  LIN {X 4999.921,Y 0.097,Z -215.600,A 90.00334,B 0.00000,C 180.00000} ; insert
  LIN {X 4999.921,Y 0.097,Z -215.600,A 90.00334,B 0.00000,C 180.00000} ; release
  LIN {X 4999.921,Y 0.097,Z 84.400,A 90.00334,B 0.00000,C 180.00000} ; retreat
  ; Step 681, bar 945
  LIN {X 5015.921,Y 0.097,Z 947.280,A 90.00334,B 0.00000,C 180.00000} ; outside
  LIN {X 5015.921,Y 0.097,Z 34.400,A 90.00334,B 0.00000,C 180.00000} ; preinsert
  LIN {X 5015.921,Y 0.097,Z -215.600,A 90.00334,B 0.00000,C 180.00000} ; insert
  LIN {X 5015.921,Y 0.097,Z -215.600,A 90.00334,B 0.00000,C 180.00000} ; release
  LIN {X 5015.921,Y 0.097,Z 84.400,A 90.00334,B 0.00000,C 180.00000} ; retreat
  ; Step 682, bar 943
  LIN {X 5124.921,Y 0.097,Z 947.280,A 90.00334,B 0.00000,C 180.00000} ; outside
  LIN {X 5124.921,Y 0.097,Z 34.400,A 90.00334,B 0.00000,C 180.00000} ; preinsert
  LIN {X 5124.921,Y 0.097,Z -215.600,A 90.00334,B 0.00000,C 180.00000} ; insert
  LIN {X 5124.921,Y 0.097,Z -215.600,A 90.00334,B 0.00000,C 180.00000} ; release
  LIN {X 5124.921,Y 0.097,Z 84.400,A 90.00334,B 0.00000,C 180.00000} ; retreat
  ; Step 683, bar 946
  LIN {X 5249.921,Y 0.097,Z 947.280,A 90.00334,B 0.00000,C 180.00000} ; outside
  LIN {X 5249.921,Y 0.097,Z 34.400,A 90.00334,B 0.00000,C 180.00000} ; preinsert
  LIN {X 5249.921,Y 0.097,Z -215.600,A 90.00334,B 0.00000,C 180.00000} ; insert
  LIN {X 5249.921,Y 0.097,Z -215.600,A 90.00334,B 0.00000,C 180.00000} ; release
  LIN {X 5249.921,Y 0.097,Z 84.400,A 90.00334,B 0.00000,C 180.00000} ; retreat
  ; Step 684, bar 947
  LIN {X 5374.921,Y 0.097,Z 947.280,A 90.00334,B 0.00000,C 180.00000} ; outside
  LIN {X 5374.921,Y 0.097,Z 34.400,A 90.00334,B 0.00000,C 180.00000} ; preinsert
  LIN {X 5374.921,Y 0.097,Z -215.600,A 90.00334,B 0.00000,C 180.00000} ; insert
  LIN {X 5374.921,Y 0.097,Z -215.600,A 90.00334,B 0.00000,C 180.00000} ; release
  LIN {X 5374.921,Y 0.097,Z 84.400,A 90.00334,B 0.00000,C 180.00000} ; retreat
  ; Step 685, bar 949
  LIN {X 5499.921,Y 0.097,Z 947.280,A 90.00334,B 0.00000,C 180.00000} ; outside
  LIN {X 5499.921,Y 0.097,Z 34.400,A 90.00334,B 0.00000,C 180.00000} ; preinsert
  LIN {X 5499.921,Y 0.097,Z -215.600,A 90.00334,B 0.00000,C 180.00000} ; insert
  LIN {X 5499.921,Y 0.097,Z -215.600,A 90.00334,B 0.00000,C 180.00000} ; release
  LIN {X 5499.921,Y 0.097,Z 84.400,A 90.00334,B 0.00000,C 180.00000} ; retreat
  ; Step 686, bar 950
  LIN {X 5515.921,Y 0.097,Z 947.280,A 90.00334,B 0.00000,C 180.00000} ; outside
  LIN {X 5515.921,Y 0.097,Z 34.400,A 90.00334,B 0.00000,C 180.00000} ; preinsert
  LIN {X 5515.921,Y 0.097,Z -215.600,A 90.00334,B 0.00000,C 180.00000} ; insert
  LIN {X 5515.921,Y 0.097,Z -215.600,A 90.00334,B 0.00000,C 180.00000} ; release
  LIN {X 5515.921,Y 0.097,Z 84.400,A 90.00334,B 0.00000,C 180.00000} ; retreat
  ; Step 687, bar 948
  LIN {X 5624.921,Y 0.097,Z 947.280,A 90.00334,B 0.00000,C 180.00000} ; outside
  LIN {X 5624.921,Y 0.097,Z 34.400,A 90.00334,B 0.00000,C 180.00000} ; preinsert
  LIN {X 5624.921,Y 0.097,Z -215.600,A 90.00334,B 0.00000,C 180.00000} ; insert
  LIN {X 5624.921,Y 0.097,Z -215.600,A 90.00334,B 0.00000,C 180.00000} ; release
  LIN {X 5624.921,Y 0.097,Z 84.400,A 90.00334,B 0.00000,C 180.00000} ; retreat
  ; Step 688, bar 951
  LIN {X 5749.921,Y 0.097,Z 947.280,A 90.00334,B 0.00000,C 180.00000} ; outside
  LIN {X 5749.921,Y 0.097,Z 34.400,A 90.00334,B 0.00000,C 180.00000} ; preinsert
  LIN {X 5749.921,Y 0.097,Z -215.600,A 90.00334,B 0.00000,C 180.00000} ; insert
  LIN {X 5749.921,Y 0.097,Z -215.600,A 90.00334,B 0.00000,C 180.00000} ; release
  LIN {X 5749.921,Y 0.097,Z 84.400,A 90.00334,B 0.00000,C 180.00000} ; retreat
  ; Step 689, bar 954
  LIN {X 5874.921,Y 0.097,Z 947.280,A 90.00334,B 0.00000,C 180.00000} ; outside
  LIN {X 5874.921,Y 0.097,Z 34.400,A 90.00334,B 0.00000,C 180.00000} ; preinsert
  LIN {X 5874.921,Y 0.097,Z -215.600,A 90.00334,B 0.00000,C 180.00000} ; insert
  LIN {X 5874.921,Y 0.097,Z -215.600,A 90.00334,B 0.00000,C 180.00000} ; release
  LIN {X 5874.921,Y 0.097,Z 84.400,A 90.00334,B 0.00000,C 180.00000} ; retreat
  ; Step 690, bar 955
  LIN {X 5890.921,Y 0.097,Z 947.280,A 90.00334,B 0.00000,C 180.00000} ; outside
  LIN {X 5890.921,Y 0.097,Z 34.400,A 90.00334,B 0.00000,C 180.00000} ; preinsert
  LIN {X 5890.921,Y 0.097,Z -215.600,A 90.00334,B 0.00000,C 180.00000} ; insert
  LIN {X 5890.921,Y 0.097,Z -215.600,A 90.00334,B 0.00000,C 180.00000} ; release
  LIN {X 5890.921,Y 0.097,Z 84.400,A 90.00334,B 0.00000,C 180.00000} ; retreat
  ; Step 691, bar 952
  LIN {X 5999.921,Y 0.097,Z 947.280,A 90.00334,B 0.00000,C 180.00000} ; outside
  LIN {X 5999.921,Y 0.097,Z 34.400,A 90.00334,B 0.00000,C 180.00000} ; preinsert
  LIN {X 5999.921,Y 0.097,Z -215.600,A 90.00334,B 0.00000,C 180.00000} ; insert
  LIN {X 5999.921,Y 0.097,Z -215.600,A 90.00334,B 0.00000,C 180.00000} ; release
  LIN {X 5999.921,Y 0.097,Z 84.400,A 90.00334,B 0.00000,C 180.00000} ; retreat
  ; Step 692, bar 953
  LIN {X 6124.921,Y 0.097,Z 947.280,A 90.00334,B 0.00000,C 180.00000} ; outside
  LIN {X 6124.921,Y 0.097,Z 34.400,A 90.00334,B 0.00000,C 180.00000} ; preinsert
  LIN {X 6124.921,Y 0.097,Z -215.600,A 90.00334,B 0.00000,C 180.00000} ; insert
  LIN {X 6124.921,Y 0.097,Z -215.600,A 90.00334,B 0.00000,C 180.00000} ; release
  LIN {X 6124.921,Y 0.097,Z 84.400,A 90.00334,B 0.00000,C 180.00000} ; retreat
  ; Step 693, bar 956
  LIN {X 6249.921,Y 0.097,Z 947.280,A 90.00334,B 0.00000,C 180.00000} ; outside
  LIN {X 6249.921,Y 0.097,Z 34.400,A 90.00334,B 0.00000,C 180.00000} ; preinsert
  LIN {X 6249.921,Y 0.097,Z -215.600,A 90.00334,B 0.00000,C 180.00000} ; insert
  LIN {X 6249.921,Y 0.097,Z -215.600,A 90.00334,B 0.00000,C 180.00000} ; release
  LIN {X 6249.921,Y 0.097,Z 84.400,A 90.00334,B 0.00000,C 180.00000} ; retreat
  ; Step 694, bar 957
  LIN {X 6374.921,Y 0.097,Z 947.280,A 90.00334,B 0.00000,C 180.00000} ; outside
  LIN {X 6374.921,Y 0.097,Z 34.400,A 90.00334,B 0.00000,C 180.00000} ; preinsert
  LIN {X 6374.921,Y 0.097,Z -215.600,A 90.00334,B 0.00000,C 180.00000} ; insert
  LIN {X 6374.921,Y 0.097,Z -215.600,A 90.00334,B 0.00000,C 180.00000} ; release
  LIN {X 6374.921,Y 0.097,Z 84.400,A 90.00334,B 0.00000,C 180.00000} ; retreat
  ; Step 695, bar 959
  LIN {X 6499.921,Y 0.097,Z 947.280,A 90.00334,B 0.00000,C 180.00000} ; outside
  LIN {X 6499.921,Y 0.097,Z 34.400,A 90.00334,B 0.00000,C 180.00000} ; preinsert
  LIN {X 6499.921,Y 0.097,Z -215.600,A 90.00334,B 0.00000,C 180.00000} ; insert
  LIN {X 6499.921,Y 0.097,Z -215.600,A 90.00334,B 0.00000,C 180.00000} ; release
  LIN {X 6499.921,Y 0.097,Z 84.400,A 90.00334,B 0.00000,C 180.00000} ; retreat
  ; Step 696, bar 960
  LIN {X 6515.921,Y 0.097,Z 947.280,A 90.00334,B 0.00000,C 180.00000} ; outside
  LIN {X 6515.921,Y 0.097,Z 34.400,A 90.00334,B 0.00000,C 180.00000} ; preinsert
  LIN {X 6515.921,Y 0.097,Z -215.600,A 90.00334,B 0.00000,C 180.00000} ; insert
  LIN {X 6515.921,Y 0.097,Z -215.600,A 90.00334,B 0.00000,C 180.00000} ; release
  LIN {X 6515.921,Y 0.097,Z 84.400,A 90.00334,B 0.00000,C 180.00000} ; retreat
  ; Step 697, bar 958
  LIN {X 6624.921,Y 0.097,Z 947.280,A 90.00334,B 0.00000,C 180.00000} ; outside
  LIN {X 6624.921,Y 0.097,Z 34.400,A 90.00334,B 0.00000,C 180.00000} ; preinsert
  LIN {X 6624.921,Y 0.097,Z -215.600,A 90.00334,B 0.00000,C 180.00000} ; insert
  LIN {X 6624.921,Y 0.097,Z -215.600,A 90.00334,B 0.00000,C 180.00000} ; release
  LIN {X 6624.921,Y 0.097,Z 84.400,A 90.00334,B 0.00000,C 180.00000} ; retreat
  ; Step 698, bar 961
  LIN {X 6749.921,Y 0.097,Z 947.280,A 90.00334,B 0.00000,C 180.00000} ; outside
  LIN {X 6749.921,Y 0.097,Z 34.400,A 90.00334,B 0.00000,C 180.00000} ; preinsert
  LIN {X 6749.921,Y 0.097,Z -215.600,A 90.00334,B 0.00000,C 180.00000} ; insert
  LIN {X 6749.921,Y 0.097,Z -215.600,A 90.00334,B 0.00000,C 180.00000} ; release
  LIN {X 6749.921,Y 0.097,Z 84.400,A 90.00334,B 0.00000,C 180.00000} ; retreat
  ; Step 699, bar 962
  LIN {X 6874.921,Y 0.097,Z 947.280,A 90.00334,B 0.00000,C 180.00000} ; outside
  LIN {X 6874.921,Y 0.097,Z 34.400,A 90.00334,B 0.00000,C 180.00000} ; preinsert
  LIN {X 6874.921,Y 0.097,Z -215.600,A 90.00334,B 0.00000,C 180.00000} ; insert
  LIN {X 6874.921,Y 0.097,Z -215.600,A 90.00334,B 0.00000,C 180.00000} ; release
  LIN {X 6874.921,Y 0.097,Z 84.400,A 90.00334,B 0.00000,C 180.00000} ; retreat
  ; Step 700, bar 964
  LIN {X 6999.921,Y 0.097,Z 947.280,A 90.00334,B 0.00000,C 180.00000} ; outside
  LIN {X 6999.921,Y 0.097,Z 34.400,A 90.00334,B 0.00000,C 180.00000} ; preinsert
  LIN {X 6999.921,Y 0.097,Z -215.600,A 90.00334,B 0.00000,C 180.00000} ; insert
  LIN {X 6999.921,Y 0.097,Z -215.600,A 90.00334,B 0.00000,C 180.00000} ; release
  LIN {X 6999.921,Y 0.097,Z 84.400,A 90.00334,B 0.00000,C 180.00000} ; retreat
  ; Step 701, bar 965
  LIN {X 7015.921,Y 0.097,Z 947.280,A 90.00334,B 0.00000,C 180.00000} ; outside
  LIN {X 7015.921,Y 0.097,Z 34.400,A 90.00334,B 0.00000,C 180.00000} ; preinsert
  LIN {X 7015.921,Y 0.097,Z -215.600,A 90.00334,B 0.00000,C 180.00000} ; insert
  LIN {X 7015.921,Y 0.097,Z -215.600,A 90.00334,B 0.00000,C 180.00000} ; release
  LIN {X 7015.921,Y 0.097,Z 84.400,A 90.00334,B 0.00000,C 180.00000} ; retreat
  ; Step 702, bar 963
  LIN {X 7124.921,Y 0.097,Z 947.280,A 90.00334,B 0.00000,C 180.00000} ; outside
  LIN {X 7124.921,Y 0.097,Z 34.400,A 90.00334,B 0.00000,C 180.00000} ; preinsert
  LIN {X 7124.921,Y 0.097,Z -215.600,A 90.00334,B 0.00000,C 180.00000} ; insert
  LIN {X 7124.921,Y 0.097,Z -215.600,A 90.00334,B 0.00000,C 180.00000} ; release
  LIN {X 7124.921,Y 0.097,Z 84.400,A 90.00334,B 0.00000,C 180.00000} ; retreat
  ; Step 703, bar 966
  LIN {X 7249.921,Y 0.097,Z 947.280,A 90.00334,B 0.00000,C 180.00000} ; outside
  LIN {X 7249.921,Y 0.097,Z 34.400,A 90.00334,B 0.00000,C 180.00000} ; preinsert
  LIN {X 7249.921,Y 0.097,Z -215.600,A 90.00334,B 0.00000,C 180.00000} ; insert
  LIN {X 7249.921,Y 0.097,Z -215.600,A 90.00334,B 0.00000,C 180.00000} ; release
  LIN {X 7249.921,Y 0.097,Z 84.400,A 90.00334,B 0.00000,C 180.00000} ; retreat
  ; Step 704, bar 967
  LIN {X 7374.921,Y 0.097,Z 947.280,A 90.00334,B 0.00000,C 180.00000} ; outside
  LIN {X 7374.921,Y 0.097,Z 34.400,A 90.00334,B 0.00000,C 180.00000} ; preinsert
  LIN {X 7374.921,Y 0.097,Z -215.600,A 90.00334,B 0.00000,C 180.00000} ; insert
  LIN {X 7374.921,Y 0.097,Z -215.600,A 90.00334,B 0.00000,C 180.00000} ; release
  LIN {X 7374.921,Y 0.097,Z 84.400,A 90.00334,B 0.00000,C 180.00000} ; retreat
  ; Step 705, bar 969
  LIN {X 7499.921,Y 0.097,Z 947.280,A 90.00334,B 0.00000,C 180.00000} ; outside
  LIN {X 7499.921,Y 0.097,Z 34.400,A 90.00334,B 0.00000,C 180.00000} ; preinsert
  LIN {X 7499.921,Y 0.097,Z -215.600,A 90.00334,B 0.00000,C 180.00000} ; insert
  LIN {X 7499.921,Y 0.097,Z -215.600,A 90.00334,B 0.00000,C 180.00000} ; release
  LIN {X 7499.921,Y 0.097,Z 84.400,A 90.00334,B 0.00000,C 180.00000} ; retreat
  ; Step 706, bar 970
  LIN {X 7515.921,Y 0.097,Z 947.280,A 90.00334,B 0.00000,C 180.00000} ; outside
  LIN {X 7515.921,Y 0.097,Z 34.400,A 90.00334,B 0.00000,C 180.00000} ; preinsert
  LIN {X 7515.921,Y 0.097,Z -215.600,A 90.00334,B 0.00000,C 180.00000} ; insert
  LIN {X 7515.921,Y 0.097,Z -215.600,A 90.00334,B 0.00000,C 180.00000} ; release
  LIN {X 7515.921,Y 0.097,Z 84.400,A 90.00334,B 0.00000,C 180.00000} ; retreat
  ; Step 707, bar 968
  LIN {X 7624.921,Y 0.097,Z 947.280,A 90.00334,B 0.00000,C 180.00000} ; outside
  LIN {X 7624.921,Y 0.097,Z 34.400,A 90.00334,B 0.00000,C 180.00000} ; preinsert
  LIN {X 7624.921,Y 0.097,Z -215.600,A 90.00334,B 0.00000,C 180.00000} ; insert
  LIN {X 7624.921,Y 0.097,Z -215.600,A 90.00334,B 0.00000,C 180.00000} ; release
  LIN {X 7624.921,Y 0.097,Z 84.400,A 90.00334,B 0.00000,C 180.00000} ; retreat
  ; Step 708, bar 971
  LIN {X 7749.921,Y 0.097,Z 947.280,A 90.00334,B 0.00000,C 180.00000} ; outside
  LIN {X 7749.921,Y 0.097,Z 34.400,A 90.00334,B 0.00000,C 180.00000} ; preinsert
  LIN {X 7749.921,Y 0.097,Z -215.600,A 90.00334,B 0.00000,C 180.00000} ; insert
  LIN {X 7749.921,Y 0.097,Z -215.600,A 90.00334,B 0.00000,C 180.00000} ; release
  LIN {X 7749.921,Y 0.097,Z 84.400,A 90.00334,B 0.00000,C 180.00000} ; retreat
  ; Step 709, bar 972
  LIN {X 7874.921,Y 0.097,Z 947.280,A 90.00334,B 0.00000,C 180.00000} ; outside
  LIN {X 7874.921,Y 0.097,Z 34.400,A 90.00334,B 0.00000,C 180.00000} ; preinsert
  LIN {X 7874.921,Y 0.097,Z -215.600,A 90.00334,B 0.00000,C 180.00000} ; insert
  LIN {X 7874.921,Y 0.097,Z -215.600,A 90.00334,B 0.00000,C 180.00000} ; release
  LIN {X 7874.921,Y 0.097,Z 84.400,A 90.00334,B 0.00000,C 180.00000} ; retreat
  ; Step 710, bar 974
  LIN {X 7999.921,Y 0.097,Z 947.280,A 90.00334,B 0.00000,C 180.00000} ; outside
  LIN {X 7999.921,Y 0.097,Z 34.400,A 90.00334,B 0.00000,C 180.00000} ; preinsert
  LIN {X 7999.921,Y 0.097,Z -215.600,A 90.00334,B 0.00000,C 180.00000} ; insert
  LIN {X 7999.921,Y 0.097,Z -215.600,A 90.00334,B 0.00000,C 180.00000} ; release
  LIN {X 7999.921,Y 0.097,Z 84.400,A 90.00334,B 0.00000,C 180.00000} ; retreat
  ; Step 711, bar 975
  LIN {X 8015.921,Y 0.097,Z 947.280,A 90.00334,B 0.00000,C 180.00000} ; outside
  LIN {X 8015.921,Y 0.097,Z 34.400,A 90.00334,B 0.00000,C 180.00000} ; preinsert
  LIN {X 8015.921,Y 0.097,Z -215.600,A 90.00334,B 0.00000,C 180.00000} ; insert
  LIN {X 8015.921,Y 0.097,Z -215.600,A 90.00334,B 0.00000,C 180.00000} ; release
  LIN {X 8015.921,Y 0.097,Z 84.400,A 90.00334,B 0.00000,C 180.00000} ; retreat
  ; Step 712, bar 973
  LIN {X 8124.921,Y 0.097,Z 947.280,A 90.00334,B 0.00000,C 180.00000} ; outside
  LIN {X 8124.921,Y 0.097,Z 34.400,A 90.00334,B 0.00000,C 180.00000} ; preinsert
  LIN {X 8124.921,Y 0.097,Z -215.600,A 90.00334,B 0.00000,C 180.00000} ; insert
  LIN {X 8124.921,Y 0.097,Z -215.600,A 90.00334,B 0.00000,C 180.00000} ; release
  LIN {X 8124.921,Y 0.097,Z 84.400,A 90.00334,B 0.00000,C 180.00000} ; retreat
  ; Step 713, bar 976
  LIN {X 8249.921,Y 0.097,Z 947.280,A 90.00334,B 0.00000,C 180.00000} ; outside
  LIN {X 8249.921,Y 0.097,Z 34.400,A 90.00334,B 0.00000,C 180.00000} ; preinsert
  LIN {X 8249.921,Y 0.097,Z -215.600,A 90.00334,B 0.00000,C 180.00000} ; insert
  LIN {X 8249.921,Y 0.097,Z -215.600,A 90.00334,B 0.00000,C 180.00000} ; release
  LIN {X 8249.921,Y 0.097,Z 84.400,A 90.00334,B 0.00000,C 180.00000} ; retreat
  ; Step 714, bar 977
  LIN {X 8374.921,Y 0.097,Z 947.280,A 90.00334,B 0.00000,C 180.00000} ; outside
  LIN {X 8374.921,Y 0.097,Z 34.400,A 90.00334,B 0.00000,C 180.00000} ; preinsert
  LIN {X 8374.921,Y 0.097,Z -215.600,A 90.00334,B 0.00000,C 180.00000} ; insert
  LIN {X 8374.921,Y 0.097,Z -215.600,A 90.00334,B 0.00000,C 180.00000} ; release
  LIN {X 8374.921,Y 0.097,Z 84.400,A 90.00334,B 0.00000,C 180.00000} ; retreat
  ; Step 715, bar 979
  LIN {X 8499.921,Y 0.097,Z 947.280,A 90.00334,B 0.00000,C 180.00000} ; outside
  LIN {X 8499.921,Y 0.097,Z 34.400,A 90.00334,B 0.00000,C 180.00000} ; preinsert
  LIN {X 8499.921,Y 0.097,Z -215.600,A 90.00334,B 0.00000,C 180.00000} ; insert
  LIN {X 8499.921,Y 0.097,Z -215.600,A 90.00334,B 0.00000,C 180.00000} ; release
  LIN {X 8499.921,Y 0.097,Z 84.400,A 90.00334,B 0.00000,C 180.00000} ; retreat
  ; Step 716, bar 980
  LIN {X 8515.921,Y 0.097,Z 947.280,A 90.00334,B 0.00000,C 180.00000} ; outside
  LIN {X 8515.921,Y 0.097,Z 34.400,A 90.00334,B 0.00000,C 180.00000} ; preinsert
  LIN {X 8515.921,Y 0.097,Z -215.600,A 90.00334,B 0.00000,C 180.00000} ; insert
  LIN {X 8515.921,Y 0.097,Z -215.600,A 90.00334,B 0.00000,C 180.00000} ; release
  LIN {X 8515.921,Y 0.097,Z 84.400,A 90.00334,B 0.00000,C 180.00000} ; retreat
  ; Step 717, bar 978
  LIN {X 8624.921,Y 0.097,Z 947.280,A 90.00334,B 0.00000,C 180.00000} ; outside
  LIN {X 8624.921,Y 0.097,Z 34.400,A 90.00334,B 0.00000,C 180.00000} ; preinsert
  LIN {X 8624.921,Y 0.097,Z -215.600,A 90.00334,B 0.00000,C 180.00000} ; insert
  LIN {X 8624.921,Y 0.097,Z -215.600,A 90.00334,B 0.00000,C 180.00000} ; release
  LIN {X 8624.921,Y 0.097,Z 84.400,A 90.00334,B 0.00000,C 180.00000} ; retreat
  ; Step 718, bar 981
  LIN {X 8749.921,Y 0.097,Z 947.280,A 90.00334,B 0.00000,C 180.00000} ; outside
  LIN {X 8749.921,Y 0.097,Z 34.400,A 90.00334,B 0.00000,C 180.00000} ; preinsert
  LIN {X 8749.921,Y 0.097,Z -215.600,A 90.00334,B 0.00000,C 180.00000} ; insert
  LIN {X 8749.921,Y 0.097,Z -215.600,A 90.00334,B 0.00000,C 180.00000} ; release
  LIN {X 8749.921,Y 0.097,Z 84.400,A 90.00334,B 0.00000,C 180.00000} ; retreat
  ; Step 719, bar 982
  LIN {X 8874.921,Y 0.097,Z 947.280,A 90.00334,B 0.00000,C 180.00000} ; outside
  LIN {X 8874.921,Y 0.097,Z 34.400,A 90.00334,B 0.00000,C 180.00000} ; preinsert
  LIN {X 8874.921,Y 0.097,Z -215.600,A 90.00334,B 0.00000,C 180.00000} ; insert
  LIN {X 8874.921,Y 0.097,Z -215.600,A 90.00334,B 0.00000,C 180.00000} ; release
  LIN {X 8874.921,Y 0.097,Z 84.400,A 90.00334,B 0.00000,C 180.00000} ; retreat
  ; Step 720, bar 984
  LIN {X 8999.921,Y 0.097,Z 947.280,A 90.00334,B 0.00000,C 180.00000} ; outside
  LIN {X 8999.921,Y 0.097,Z 34.400,A 90.00334,B 0.00000,C 180.00000} ; preinsert
  LIN {X 8999.921,Y 0.097,Z -215.600,A 90.00334,B 0.00000,C 180.00000} ; insert
  LIN {X 8999.921,Y 0.097,Z -215.600,A 90.00334,B 0.00000,C 180.00000} ; release
  LIN {X 8999.921,Y 0.097,Z 84.400,A 90.00334,B 0.00000,C 180.00000} ; retreat
  ; Step 721, bar 985
  LIN {X 9015.921,Y 0.097,Z 947.280,A 90.00334,B 0.00000,C 180.00000} ; outside
  LIN {X 9015.921,Y 0.097,Z 34.400,A 90.00334,B 0.00000,C 180.00000} ; preinsert
  LIN {X 9015.921,Y 0.097,Z -215.600,A 90.00334,B 0.00000,C 180.00000} ; insert
  LIN {X 9015.921,Y 0.097,Z -215.600,A 90.00334,B 0.00000,C 180.00000} ; release
  LIN {X 9015.921,Y 0.097,Z 84.400,A 90.00334,B 0.00000,C 180.00000} ; retreat
  ; Step 722, bar 983
  LIN {X 9124.921,Y 0.097,Z 947.280,A 90.00334,B 0.00000,C 180.00000} ; outside
  LIN {X 9124.921,Y 0.097,Z 34.400,A 90.00334,B 0.00000,C 180.00000} ; preinsert
  LIN {X 9124.921,Y 0.097,Z -215.600,A 90.00334,B 0.00000,C 180.00000} ; insert
  LIN {X 9124.921,Y 0.097,Z -215.600,A 90.00334,B 0.00000,C 180.00000} ; release
  LIN {X 9124.921,Y 0.097,Z 84.400,A 90.00334,B 0.00000,C 180.00000} ; retreat
  ; Step 723, bar 986
  LIN {X 9249.921,Y 0.097,Z 947.280,A 90.00334,B 0.00000,C 180.00000} ; outside
  LIN {X 9249.921,Y 0.097,Z 34.400,A 90.00334,B 0.00000,C 180.00000} ; preinsert
  LIN {X 9249.921,Y 0.097,Z -215.600,A 90.00334,B 0.00000,C 180.00000} ; insert
  LIN {X 9249.921,Y 0.097,Z -215.600,A 90.00334,B 0.00000,C 180.00000} ; release
  LIN {X 9249.921,Y 0.097,Z 84.400,A 90.00334,B 0.00000,C 180.00000} ; retreat
  ; Step 724, bar 987
  LIN {X 9374.921,Y 0.097,Z 947.280,A 90.00334,B 0.00000,C 180.00000} ; outside
  LIN {X 9374.921,Y 0.097,Z 34.400,A 90.00334,B 0.00000,C 180.00000} ; preinsert
  LIN {X 9374.921,Y 0.097,Z -215.600,A 90.00334,B 0.00000,C 180.00000} ; insert
  LIN {X 9374.921,Y 0.097,Z -215.600,A 90.00334,B 0.00000,C 180.00000} ; release
  LIN {X 9374.921,Y 0.097,Z 84.400,A 90.00334,B 0.00000,C 180.00000} ; retreat
  ; Step 725, bar 989
  LIN {X 9499.921,Y 0.097,Z 947.280,A 90.00334,B 0.00000,C 180.00000} ; outside
  LIN {X 9499.921,Y 0.097,Z 34.400,A 90.00334,B 0.00000,C 180.00000} ; preinsert
  LIN {X 9499.921,Y 0.097,Z -215.600,A 90.00334,B 0.00000,C 180.00000} ; insert
  LIN {X 9499.921,Y 0.097,Z -215.600,A 90.00334,B 0.00000,C 180.00000} ; release
  LIN {X 9499.921,Y 0.097,Z 84.400,A 90.00334,B 0.00000,C 180.00000} ; retreat
  ; Step 726, bar 990
  LIN {X 9515.921,Y 0.097,Z 947.280,A 90.00334,B 0.00000,C 180.00000} ; outside
  LIN {X 9515.921,Y 0.097,Z 34.400,A 90.00334,B 0.00000,C 180.00000} ; preinsert
  LIN {X 9515.921,Y 0.097,Z -215.600,A 90.00334,B 0.00000,C 180.00000} ; insert
  LIN {X 9515.921,Y 0.097,Z -215.600,A 90.00334,B 0.00000,C 180.00000} ; release
  LIN {X 9515.921,Y 0.097,Z 84.400,A 90.00334,B 0.00000,C 180.00000} ; retreat
  ; Step 727, bar 988
  LIN {X 9624.921,Y 0.097,Z 947.280,A 90.00334,B 0.00000,C 180.00000} ; outside
  LIN {X 9624.921,Y 0.097,Z 34.400,A 90.00334,B 0.00000,C 180.00000} ; preinsert
  LIN {X 9624.921,Y 0.097,Z -215.600,A 90.00334,B 0.00000,C 180.00000} ; insert
  LIN {X 9624.921,Y 0.097,Z -215.600,A 90.00334,B 0.00000,C 180.00000} ; release
  LIN {X 9624.921,Y 0.097,Z 84.400,A 90.00334,B 0.00000,C 180.00000} ; retreat
  ; Step 728, bar 991
  LIN {X 9749.921,Y 0.097,Z 947.280,A 90.00334,B 0.00000,C 180.00000} ; outside
  LIN {X 9749.921,Y 0.097,Z 34.400,A 90.00334,B 0.00000,C 180.00000} ; preinsert
  LIN {X 9749.921,Y 0.097,Z -215.600,A 90.00334,B 0.00000,C 180.00000} ; insert
  LIN {X 9749.921,Y 0.097,Z -215.600,A 90.00334,B 0.00000,C 180.00000} ; release
  LIN {X 9749.921,Y 0.097,Z 84.400,A 90.00334,B 0.00000,C 180.00000} ; retreat
  ; Step 729, bar 994
  LIN {X 9874.921,Y 0.097,Z 947.280,A 90.00334,B 0.00000,C 180.00000} ; outside
  LIN {X 9874.921,Y 0.097,Z 34.400,A 90.00334,B 0.00000,C 180.00000} ; preinsert
  LIN {X 9874.921,Y 0.097,Z -215.600,A 90.00334,B 0.00000,C 180.00000} ; insert
  LIN {X 9874.921,Y 0.097,Z -215.600,A 90.00334,B 0.00000,C 180.00000} ; release
  LIN {X 9874.921,Y 0.097,Z 84.400,A 90.00334,B 0.00000,C 180.00000} ; retreat
  ; Step 730, bar 995
  LIN {X 9890.921,Y 0.097,Z 947.280,A 90.00334,B 0.00000,C 180.00000} ; outside
  LIN {X 9890.921,Y 0.097,Z 34.400,A 90.00334,B 0.00000,C 180.00000} ; preinsert
  LIN {X 9890.921,Y 0.097,Z -215.600,A 90.00334,B 0.00000,C 180.00000} ; insert
  LIN {X 9890.921,Y 0.097,Z -215.600,A 90.00334,B 0.00000,C 180.00000} ; release
  LIN {X 9890.921,Y 0.097,Z 84.400,A 90.00334,B 0.00000,C 180.00000} ; retreat
  ; Step 731, bar 992
  LIN {X 9999.921,Y 0.097,Z 947.280,A 90.00334,B 0.00000,C 180.00000} ; outside
  LIN {X 9999.921,Y 0.097,Z 34.400,A 90.00334,B 0.00000,C 180.00000} ; preinsert
  LIN {X 9999.921,Y 0.097,Z -215.600,A 90.00334,B 0.00000,C 180.00000} ; insert
  LIN {X 9999.921,Y 0.097,Z -215.600,A 90.00334,B 0.00000,C 180.00000} ; release
  LIN {X 9999.921,Y 0.097,Z 84.400,A 90.00334,B 0.00000,C 180.00000} ; retreat
  ; Step 732, bar 993
  LIN {X 10124.921,Y 0.097,Z 947.280,A 90.00334,B 0.00000,C 180.00000} ; outside
  LIN {X 10124.921,Y 0.097,Z 34.400,A 90.00334,B 0.00000,C 180.00000} ; preinsert
  LIN {X 10124.921,Y 0.097,Z -215.600,A 90.00334,B 0.00000,C 180.00000} ; insert
  LIN {X 10124.921,Y 0.097,Z -215.600,A 90.00334,B 0.00000,C 180.00000} ; release
  LIN {X 10124.921,Y 0.097,Z 84.400,A 90.00334,B 0.00000,C 180.00000} ; retreat
  ; Step 733, bar 996
  LIN {X 10249.921,Y 0.097,Z 947.280,A 90.00334,B 0.00000,C 180.00000} ; outside
  LIN {X 10249.921,Y 0.097,Z 34.400,A 90.00334,B 0.00000,C 180.00000} ; preinsert
  LIN {X 10249.921,Y 0.097,Z -215.600,A 90.00334,B 0.00000,C 180.00000} ; insert
  LIN {X 10249.921,Y 0.097,Z -215.600,A 90.00334,B 0.00000,C 180.00000} ; release
  LIN {X 10249.921,Y 0.097,Z 84.400,A 90.00334,B 0.00000,C 180.00000} ; retreat
  ; Step 734, bar 997
  LIN {X 10374.921,Y 0.097,Z 947.280,A 90.00334,B 0.00000,C 180.00000} ; outside
  LIN {X 10374.921,Y 0.097,Z 34.400,A 90.00334,B 0.00000,C 180.00000} ; preinsert
  LIN {X 10374.921,Y 0.097,Z -215.600,A 90.00334,B 0.00000,C 180.00000} ; insert
  LIN {X 10374.921,Y 0.097,Z -215.600,A 90.00334,B 0.00000,C 180.00000} ; release
  LIN {X 10374.921,Y 0.097,Z 84.400,A 90.00334,B 0.00000,C 180.00000} ; retreat
  ; Step 735, bar 999
  LIN {X 10499.921,Y 0.097,Z 947.280,A 90.00334,B 0.00000,C 180.00000} ; outside
  LIN {X 10499.921,Y 0.097,Z 34.400,A 90.00334,B 0.00000,C 180.00000} ; preinsert
  LIN {X 10499.921,Y 0.097,Z -215.600,A 90.00334,B 0.00000,C 180.00000} ; insert
  LIN {X 10499.921,Y 0.097,Z -215.600,A 90.00334,B 0.00000,C 180.00000} ; release
  LIN {X 10499.921,Y 0.097,Z 84.400,A 90.00334,B 0.00000,C 180.00000} ; retreat
  ; Step 736, bar 1000
  LIN {X 10515.921,Y 0.097,Z 947.280,A 90.00334,B 0.00000,C 180.00000} ; outside
  LIN {X 10515.921,Y 0.097,Z 34.400,A 90.00334,B 0.00000,C 180.00000} ; preinsert
  LIN {X 10515.921,Y 0.097,Z -215.600,A 90.00334,B 0.00000,C 180.00000} ; insert
  LIN {X 10515.921,Y 0.097,Z -215.600,A 90.00334,B 0.00000,C 180.00000} ; release
  LIN {X 10515.921,Y 0.097,Z 84.400,A 90.00334,B 0.00000,C 180.00000} ; retreat
  ; Step 737, bar 998
  LIN {X 10624.921,Y 0.097,Z 947.280,A 90.00334,B 0.00000,C 180.00000} ; outside
  LIN {X 10624.921,Y 0.097,Z 34.400,A 90.00334,B 0.00000,C 180.00000} ; preinsert
  LIN {X 10624.921,Y 0.097,Z -215.600,A 90.00334,B 0.00000,C 180.00000} ; insert
  LIN {X 10624.921,Y 0.097,Z -215.600,A 90.00334,B 0.00000,C 180.00000} ; release
  LIN {X 10624.921,Y 0.097,Z 84.400,A 90.00334,B 0.00000,C 180.00000} ; retreat
  ; Step 738, bar 1001
  LIN {X 10749.921,Y 0.097,Z 947.280,A 90.00334,B 0.00000,C 180.00000} ; outside
  LIN {X 10749.921,Y 0.097,Z 34.400,A 90.00334,B 0.00000,C 180.00000} ; preinsert
  LIN {X 10749.921,Y 0.097,Z -215.600,A 90.00334,B 0.00000,C 180.00000} ; insert
  LIN {X 10749.921,Y 0.097,Z -215.600,A 90.00334,B 0.00000,C 180.00000} ; release
  LIN {X 10749.921,Y 0.097,Z 84.400,A 90.00334,B 0.00000,C 180.00000} ; retreat
  ; Step 739, bar 1002
  LIN {X 10874.921,Y 0.097,Z 947.280,A 90.00334,B 0.00000,C 180.00000} ; outside
  LIN {X 10874.921,Y 0.097,Z 34.400,A 90.00334,B 0.00000,C 180.00000} ; preinsert
  LIN {X 10874.921,Y 0.097,Z -215.600,A 90.00334,B 0.00000,C 180.00000} ; insert
  LIN {X 10874.921,Y 0.097,Z -215.600,A 90.00334,B 0.00000,C 180.00000} ; release
  LIN {X 10874.921,Y 0.097,Z 84.400,A 90.00334,B 0.00000,C 180.00000} ; retreat
  ; Step 740, bar 1004
  LIN {X 10999.921,Y 0.097,Z 947.280,A 90.00334,B 0.00000,C 180.00000} ; outside
  LIN {X 10999.921,Y 0.097,Z 34.400,A 90.00334,B 0.00000,C 180.00000} ; preinsert
  LIN {X 10999.921,Y 0.097,Z -215.600,A 90.00334,B 0.00000,C 180.00000} ; insert
  LIN {X 10999.921,Y 0.097,Z -215.600,A 90.00334,B 0.00000,C 180.00000} ; release
  LIN {X 10999.921,Y 0.097,Z 84.400,A 90.00334,B 0.00000,C 180.00000} ; retreat
  ; Step 741, bar 1005
  LIN {X 11015.921,Y 0.097,Z 947.280,A 90.00334,B 0.00000,C 180.00000} ; outside
  LIN {X 11015.921,Y 0.097,Z 34.400,A 90.00334,B 0.00000,C 180.00000} ; preinsert
  LIN {X 11015.921,Y 0.097,Z -215.600,A 90.00334,B 0.00000,C 180.00000} ; insert
  LIN {X 11015.921,Y 0.097,Z -215.600,A 90.00334,B 0.00000,C 180.00000} ; release
  LIN {X 11015.921,Y 0.097,Z 84.400,A 90.00334,B 0.00000,C 180.00000} ; retreat
  ; Step 742, bar 1003
  LIN {X 11124.921,Y 0.097,Z 947.280,A 90.00334,B 0.00000,C 180.00000} ; outside
  LIN {X 11124.921,Y 0.097,Z 34.400,A 90.00334,B 0.00000,C 180.00000} ; preinsert
  LIN {X 11124.921,Y 0.097,Z -215.600,A 90.00334,B 0.00000,C 180.00000} ; insert
  LIN {X 11124.921,Y 0.097,Z -215.600,A 90.00334,B 0.00000,C 180.00000} ; release
  LIN {X 11124.921,Y 0.097,Z 84.400,A 90.00334,B 0.00000,C 180.00000} ; retreat
  ; Step 743, bar 1006
  LIN {X 11249.921,Y 0.097,Z 947.280,A 90.00334,B 0.00000,C 180.00000} ; outside
  LIN {X 11249.921,Y 0.097,Z 34.400,A 90.00334,B 0.00000,C 180.00000} ; preinsert
  LIN {X 11249.921,Y 0.097,Z -215.600,A 90.00334,B 0.00000,C 180.00000} ; insert
  LIN {X 11249.921,Y 0.097,Z -215.600,A 90.00334,B 0.00000,C 180.00000} ; release
  LIN {X 11249.921,Y 0.097,Z 84.400,A 90.00334,B 0.00000,C 180.00000} ; retreat
  ; Step 744, bar 1007
  LIN {X 11374.921,Y 0.097,Z 947.280,A 90.00334,B 0.00000,C 180.00000} ; outside
  LIN {X 11374.921,Y 0.097,Z 34.400,A 90.00334,B 0.00000,C 180.00000} ; preinsert
  LIN {X 11374.921,Y 0.097,Z -215.600,A 90.00334,B 0.00000,C 180.00000} ; insert
  LIN {X 11374.921,Y 0.097,Z -215.600,A 90.00334,B 0.00000,C 180.00000} ; release
  LIN {X 11374.921,Y 0.097,Z 84.400,A 90.00334,B 0.00000,C 180.00000} ; retreat
  ; Step 745, bar 1009
  LIN {X 11499.921,Y 0.097,Z 947.280,A 90.00334,B 0.00000,C 180.00000} ; outside
  LIN {X 11499.921,Y 0.097,Z 34.400,A 90.00334,B 0.00000,C 180.00000} ; preinsert
  LIN {X 11499.921,Y 0.097,Z -215.600,A 90.00334,B 0.00000,C 180.00000} ; insert
  LIN {X 11499.921,Y 0.097,Z -215.600,A 90.00334,B 0.00000,C 180.00000} ; release
  LIN {X 11499.921,Y 0.097,Z 84.400,A 90.00334,B 0.00000,C 180.00000} ; retreat
  ; Step 746, bar 1010
  LIN {X 11515.921,Y 0.097,Z 947.280,A 90.00334,B 0.00000,C 180.00000} ; outside
  LIN {X 11515.921,Y 0.097,Z 34.400,A 90.00334,B 0.00000,C 180.00000} ; preinsert
  LIN {X 11515.921,Y 0.097,Z -215.600,A 90.00334,B 0.00000,C 180.00000} ; insert
  LIN {X 11515.921,Y 0.097,Z -215.600,A 90.00334,B 0.00000,C 180.00000} ; release
  LIN {X 11515.921,Y 0.097,Z 84.400,A 90.00334,B 0.00000,C 180.00000} ; retreat
  ; Step 747, bar 1008
  LIN {X 11624.921,Y 0.097,Z 947.280,A 90.00334,B 0.00000,C 180.00000} ; outside
  LIN {X 11624.921,Y 0.097,Z 34.400,A 90.00334,B 0.00000,C 180.00000} ; preinsert
  LIN {X 11624.921,Y 0.097,Z -215.600,A 90.00334,B 0.00000,C 180.00000} ; insert
  LIN {X 11624.921,Y 0.097,Z -215.600,A 90.00334,B 0.00000,C 180.00000} ; release
  LIN {X 11624.921,Y 0.097,Z 84.400,A 90.00334,B 0.00000,C 180.00000} ; retreat
  ; Step 748, bar 1011
  LIN {X 11749.921,Y 0.097,Z 947.280,A 90.00334,B 0.00000,C 180.00000} ; outside
  LIN {X 11749.921,Y 0.097,Z 34.400,A 90.00334,B 0.00000,C 180.00000} ; preinsert
  LIN {X 11749.921,Y 0.097,Z -215.600,A 90.00334,B 0.00000,C 180.00000} ; insert
  LIN {X 11749.921,Y 0.097,Z -215.600,A 90.00334,B 0.00000,C 180.00000} ; release
  LIN {X 11749.921,Y 0.097,Z 84.400,A 90.00334,B 0.00000,C 180.00000} ; retreat
  ; Step 749, bar 1012
  LIN {X 11874.921,Y 0.097,Z 947.280,A 90.00334,B 0.00000,C 180.00000} ; outside
  LIN {X 11874.921,Y 0.097,Z 34.400,A 90.00334,B 0.00000,C 180.00000} ; preinsert
  LIN {X 11874.921,Y 0.097,Z -215.600,A 90.00334,B 0.00000,C 180.00000} ; insert
  LIN {X 11874.921,Y 0.097,Z -215.600,A 90.00334,B 0.00000,C 180.00000} ; release
  LIN {X 11874.921,Y 0.097,Z 84.400,A 90.00334,B 0.00000,C 180.00000} ; retreat
  ; Step 750, bar 1014
  LIN {X 11999.921,Y 0.097,Z 947.280,A 90.00334,B 0.00000,C 180.00000} ; outside
  LIN {X 11999.921,Y 0.097,Z 34.400,A 90.00334,B 0.00000,C 180.00000} ; preinsert
  LIN {X 11999.921,Y 0.097,Z -215.600,A 90.00334,B 0.00000,C 180.00000} ; insert
  LIN {X 11999.921,Y 0.097,Z -215.600,A 90.00334,B 0.00000,C 180.00000} ; release
  LIN {X 11999.921,Y 0.097,Z 84.400,A 90.00334,B 0.00000,C 180.00000} ; retreat
  ; Step 751, bar 1015
  LIN {X 12015.921,Y 0.097,Z 947.280,A 90.00334,B 0.00000,C 180.00000} ; outside
  LIN {X 12015.921,Y 0.097,Z 34.400,A 90.00334,B 0.00000,C 180.00000} ; preinsert
  LIN {X 12015.921,Y 0.097,Z -215.600,A 90.00334,B 0.00000,C 180.00000} ; insert
  LIN {X 12015.921,Y 0.097,Z -215.600,A 90.00334,B 0.00000,C 180.00000} ; release
  LIN {X 12015.921,Y 0.097,Z 84.400,A 90.00334,B 0.00000,C 180.00000} ; retreat
  ; Step 752, bar 1013
  LIN {X 12124.921,Y 0.097,Z 947.280,A 90.00334,B 0.00000,C 180.00000} ; outside
  LIN {X 12124.921,Y 0.097,Z 34.400,A 90.00334,B 0.00000,C 180.00000} ; preinsert
  LIN {X 12124.921,Y 0.097,Z -215.600,A 90.00334,B 0.00000,C 180.00000} ; insert
  LIN {X 12124.921,Y 0.097,Z -215.600,A 90.00334,B 0.00000,C 180.00000} ; release
  LIN {X 12124.921,Y 0.097,Z 84.400,A 90.00334,B 0.00000,C 180.00000} ; retreat
  ; Step 753, bar 1016
  LIN {X 12249.921,Y 0.097,Z 947.280,A 90.00334,B 0.00000,C 180.00000} ; outside
  LIN {X 12249.921,Y 0.097,Z 34.400,A 90.00334,B 0.00000,C 180.00000} ; preinsert
  LIN {X 12249.921,Y 0.097,Z -215.600,A 90.00334,B 0.00000,C 180.00000} ; insert
  LIN {X 12249.921,Y 0.097,Z -215.600,A 90.00334,B 0.00000,C 180.00000} ; release
  LIN {X 12249.921,Y 0.097,Z 84.400,A 90.00334,B 0.00000,C 180.00000} ; retreat
  ; Step 754, bar 290
  LIN {X 0.000,Y -1540.000,Z 1076.871,A 0.00000,B 0.00000,C 180.00000} ; outside
  LIN {X 0.000,Y -1540.000,Z 162.746,A 0.00000,B 0.00000,C 180.00000} ; preinsert
  LIN {X 0.000,Y -1540.000,Z -87.254,A 0.00000,B 0.00000,C 180.00000} ; insert
  LIN {X 0.000,Y -1540.000,Z -87.254,A 0.00000,B 0.00000,C 180.00000} ; release
  LIN {X 0.000,Y -1540.000,Z 212.746,A 0.00000,B 0.00000,C 180.00000} ; retreat
  ; Step 755, bar 317
  LIN {X 0.000,Y 1540.000,Z 1076.871,A 0.00000,B 0.00000,C 180.00000} ; outside
  LIN {X 0.000,Y 1540.000,Z 162.746,A 0.00000,B 0.00000,C 180.00000} ; preinsert
  LIN {X 0.000,Y 1540.000,Z -87.254,A 0.00000,B 0.00000,C 180.00000} ; insert
  LIN {X 0.000,Y 1540.000,Z -87.254,A 0.00000,B 0.00000,C 180.00000} ; release
  LIN {X 0.000,Y 1540.000,Z 212.746,A 0.00000,B 0.00000,C 180.00000} ; retreat
  ; Step 756, bar 1097
  LIN {X -14079.461,Y -1499.888,Z 868.364,A 179.99901,B 0.00000,C -180.00000} ; outside
  LIN {X -14079.461,Y -1499.888,Z -75.930,A 179.99901,B 0.00000,C -180.00000} ; preinsert
  LIN {X -14079.461,Y -1499.888,Z -325.930,A 179.99901,B 0.00000,C -180.00000} ; insert
  LIN {X -14079.461,Y -1499.888,Z -325.930,A 179.99901,B 0.00000,C -180.00000} ; release
  LIN {X -14079.461,Y -1499.888,Z -25.930,A 179.99901,B 0.00000,C -180.00000} ; retreat
  ; Step 757, bar 1076
  LIN {X 14079.461,Y -1499.888,Z 868.364,A 0.00099,B 0.00000,C 180.00000} ; outside
  LIN {X 14079.461,Y -1499.888,Z -75.930,A 0.00099,B 0.00000,C 180.00000} ; preinsert
  LIN {X 14079.461,Y -1499.888,Z -325.930,A 0.00099,B 0.00000,C 180.00000} ; insert
  LIN {X 14079.461,Y -1499.888,Z -325.930,A 0.00099,B 0.00000,C 180.00000} ; release
  LIN {X 14079.461,Y -1499.888,Z -25.930,A 0.00099,B 0.00000,C 180.00000} ; retreat
  ; Step 758, bar 1096
  LIN {X -14079.461,Y -1374.888,Z 868.364,A 179.99901,B 0.00000,C -180.00000} ; outside
  LIN {X -14079.461,Y -1374.888,Z -75.930,A 179.99901,B 0.00000,C -180.00000} ; preinsert
  LIN {X -14079.461,Y -1374.888,Z -325.930,A 179.99901,B 0.00000,C -180.00000} ; insert
  LIN {X -14079.461,Y -1374.888,Z -325.930,A 179.99901,B 0.00000,C -180.00000} ; release
  LIN {X -14079.461,Y -1374.888,Z -25.930,A 179.99901,B 0.00000,C -180.00000} ; retreat
  ; Step 759, bar 1075
  LIN {X 14079.461,Y -1374.888,Z 868.364,A 0.00099,B 0.00000,C 180.00000} ; outside
  LIN {X 14079.461,Y -1374.888,Z -75.930,A 0.00099,B 0.00000,C 180.00000} ; preinsert
  LIN {X 14079.461,Y -1374.888,Z -325.930,A 0.00099,B 0.00000,C 180.00000} ; insert
  LIN {X 14079.461,Y -1374.888,Z -325.930,A 0.00099,B 0.00000,C 180.00000} ; release
  LIN {X 14079.461,Y -1374.888,Z -25.930,A 0.00099,B 0.00000,C 180.00000} ; retreat
  ; Step 760, bar 1095
  LIN {X -14079.461,Y -1049.888,Z 868.364,A 179.99901,B 0.00000,C -180.00000} ; outside
  LIN {X -14079.461,Y -1049.888,Z -75.930,A 179.99901,B 0.00000,C -180.00000} ; preinsert
  LIN {X -14079.461,Y -1049.888,Z -325.930,A 179.99901,B 0.00000,C -180.00000} ; insert
  LIN {X -14079.461,Y -1049.888,Z -325.930,A 179.99901,B 0.00000,C -180.00000} ; release
  LIN {X -14079.461,Y -1049.888,Z -25.930,A 179.99901,B 0.00000,C -180.00000} ; retreat
  ; Step 761, bar 1072
  LIN {X 14079.461,Y -1049.888,Z 868.364,A 0.00099,B 0.00000,C 180.00000} ; outside
  LIN {X 14079.461,Y -1049.888,Z -75.930,A 0.00099,B 0.00000,C 180.00000} ; preinsert
  LIN {X 14079.461,Y -1049.888,Z -325.930,A 0.00099,B 0.00000,C 180.00000} ; insert
  LIN {X 14079.461,Y -1049.888,Z -325.930,A 0.00099,B 0.00000,C 180.00000} ; release
  LIN {X 14079.461,Y -1049.888,Z -25.930,A 0.00099,B 0.00000,C 180.00000} ; retreat
  ; Step 762, bar 1094
  LIN {X -14079.461,Y -899.888,Z 868.364,A 179.99901,B 0.00000,C -180.00000} ; outside
  LIN {X -14079.461,Y -899.888,Z -75.930,A 179.99901,B 0.00000,C -180.00000} ; preinsert
  LIN {X -14079.461,Y -899.888,Z -325.930,A 179.99901,B 0.00000,C -180.00000} ; insert
  LIN {X -14079.461,Y -899.888,Z -325.930,A 179.99901,B 0.00000,C -180.00000} ; release
  LIN {X -14079.461,Y -899.888,Z -25.930,A 179.99901,B 0.00000,C -180.00000} ; retreat
  ; Step 763, bar 1071
  LIN {X 14079.461,Y -899.888,Z 868.364,A 0.00099,B 0.00000,C 180.00000} ; outside
  LIN {X 14079.461,Y -899.888,Z -75.930,A 0.00099,B 0.00000,C 180.00000} ; preinsert
  LIN {X 14079.461,Y -899.888,Z -325.930,A 0.00099,B 0.00000,C 180.00000} ; insert
  LIN {X 14079.461,Y -899.888,Z -325.930,A 0.00099,B 0.00000,C 180.00000} ; release
  LIN {X 14079.461,Y -899.888,Z -25.930,A 0.00099,B 0.00000,C 180.00000} ; retreat
  ; Step 764, bar 1093
  LIN {X -14079.461,Y -749.888,Z 868.364,A 179.99901,B 0.00000,C -180.00000} ; outside
  LIN {X -14079.461,Y -749.888,Z -75.930,A 179.99901,B 0.00000,C -180.00000} ; preinsert
  LIN {X -14079.461,Y -749.888,Z -325.930,A 179.99901,B 0.00000,C -180.00000} ; insert
  LIN {X -14079.461,Y -749.888,Z -325.930,A 179.99901,B 0.00000,C -180.00000} ; release
  LIN {X -14079.461,Y -749.888,Z -25.930,A 179.99901,B 0.00000,C -180.00000} ; retreat
  ; Step 765, bar 1070
  LIN {X 14079.461,Y -749.888,Z 868.364,A 0.00099,B 0.00000,C 180.00000} ; outside
  LIN {X 14079.461,Y -749.888,Z -75.930,A 0.00099,B 0.00000,C 180.00000} ; preinsert
  LIN {X 14079.461,Y -749.888,Z -325.930,A 0.00099,B 0.00000,C 180.00000} ; insert
  LIN {X 14079.461,Y -749.888,Z -325.930,A 0.00099,B 0.00000,C 180.00000} ; release
  LIN {X 14079.461,Y -749.888,Z -25.930,A 0.00099,B 0.00000,C 180.00000} ; retreat
  ; Step 766, bar 1092
  LIN {X -14079.461,Y -599.888,Z 868.364,A 179.99901,B 0.00000,C -180.00000} ; outside
  LIN {X -14079.461,Y -599.888,Z -75.930,A 179.99901,B 0.00000,C -180.00000} ; preinsert
  LIN {X -14079.461,Y -599.888,Z -325.930,A 179.99901,B 0.00000,C -180.00000} ; insert
  LIN {X -14079.461,Y -599.888,Z -325.930,A 179.99901,B 0.00000,C -180.00000} ; release
  LIN {X -14079.461,Y -599.888,Z -25.930,A 179.99901,B 0.00000,C -180.00000} ; retreat
  ; Step 767, bar 1069
  LIN {X 14079.461,Y -599.888,Z 868.364,A 0.00099,B 0.00000,C 180.00000} ; outside
  LIN {X 14079.461,Y -599.888,Z -75.930,A 0.00099,B 0.00000,C 180.00000} ; preinsert
  LIN {X 14079.461,Y -599.888,Z -325.930,A 0.00099,B 0.00000,C 180.00000} ; insert
  LIN {X 14079.461,Y -599.888,Z -325.930,A 0.00099,B 0.00000,C 180.00000} ; release
  LIN {X 14079.461,Y -599.888,Z -25.930,A 0.00099,B 0.00000,C 180.00000} ; retreat
  ; Step 768, bar 1091
  LIN {X -14079.461,Y -449.888,Z 868.364,A 179.99901,B 0.00000,C -180.00000} ; outside
  LIN {X -14079.461,Y -449.888,Z -75.930,A 179.99901,B 0.00000,C -180.00000} ; preinsert
  LIN {X -14079.461,Y -449.888,Z -325.930,A 179.99901,B 0.00000,C -180.00000} ; insert
  LIN {X -14079.461,Y -449.888,Z -325.930,A 179.99901,B 0.00000,C -180.00000} ; release
  LIN {X -14079.461,Y -449.888,Z -25.930,A 179.99901,B 0.00000,C -180.00000} ; retreat
  ; Step 769, bar 1068
  LIN {X 14079.461,Y -449.888,Z 868.364,A 0.00099,B 0.00000,C 180.00000} ; outside
  LIN {X 14079.461,Y -449.888,Z -75.930,A 0.00099,B 0.00000,C 180.00000} ; preinsert
  LIN {X 14079.461,Y -449.888,Z -325.930,A 0.00099,B 0.00000,C 180.00000} ; insert
  LIN {X 14079.461,Y -449.888,Z -325.930,A 0.00099,B 0.00000,C 180.00000} ; release
  LIN {X 14079.461,Y -449.888,Z -25.930,A 0.00099,B 0.00000,C 180.00000} ; retreat
  ; Step 770, bar 1090
  LIN {X -14079.461,Y -299.888,Z 868.364,A 179.99901,B 0.00000,C -180.00000} ; outside
  LIN {X -14079.461,Y -299.888,Z -75.930,A 179.99901,B 0.00000,C -180.00000} ; preinsert
  LIN {X -14079.461,Y -299.888,Z -325.930,A 179.99901,B 0.00000,C -180.00000} ; insert
  LIN {X -14079.461,Y -299.888,Z -325.930,A 179.99901,B 0.00000,C -180.00000} ; release
  LIN {X -14079.461,Y -299.888,Z -25.930,A 179.99901,B 0.00000,C -180.00000} ; retreat
  ; Step 771, bar 1067
  LIN {X 14079.461,Y -299.888,Z 868.364,A 0.00099,B 0.00000,C 180.00000} ; outside
  LIN {X 14079.461,Y -299.888,Z -75.930,A 0.00099,B 0.00000,C 180.00000} ; preinsert
  LIN {X 14079.461,Y -299.888,Z -325.930,A 0.00099,B 0.00000,C 180.00000} ; insert
  LIN {X 14079.461,Y -299.888,Z -325.930,A 0.00099,B 0.00000,C 180.00000} ; release
  LIN {X 14079.461,Y -299.888,Z -25.930,A 0.00099,B 0.00000,C 180.00000} ; retreat
  ; Step 772, bar 1089
  LIN {X -14079.461,Y -149.888,Z 868.364,A 179.99901,B 0.00000,C -180.00000} ; outside
  LIN {X -14079.461,Y -149.888,Z -75.930,A 179.99901,B 0.00000,C -180.00000} ; preinsert
  LIN {X -14079.461,Y -149.888,Z -325.930,A 179.99901,B 0.00000,C -180.00000} ; insert
  LIN {X -14079.461,Y -149.888,Z -325.930,A 179.99901,B 0.00000,C -180.00000} ; release
  LIN {X -14079.461,Y -149.888,Z -25.930,A 179.99901,B 0.00000,C -180.00000} ; retreat
  ; Step 773, bar 1066
  LIN {X 14079.461,Y -149.888,Z 868.364,A 0.00099,B 0.00000,C 180.00000} ; outside
  LIN {X 14079.461,Y -149.888,Z -75.930,A 0.00099,B 0.00000,C 180.00000} ; preinsert
  LIN {X 14079.461,Y -149.888,Z -325.930,A 0.00099,B 0.00000,C 180.00000} ; insert
  LIN {X 14079.461,Y -149.888,Z -325.930,A 0.00099,B 0.00000,C 180.00000} ; release
  LIN {X 14079.461,Y -149.888,Z -25.930,A 0.00099,B 0.00000,C 180.00000} ; retreat
  ; Step 774, bar 1017
  LIN {X 14079.461,Y 0.112,Z 868.364,A 0.00099,B 0.00000,C 180.00000} ; outside
  LIN {X 14079.461,Y 0.112,Z -75.930,A 0.00099,B 0.00000,C 180.00000} ; preinsert
  LIN {X 14079.461,Y 0.112,Z -325.930,A 0.00099,B 0.00000,C 180.00000} ; insert
  LIN {X 14079.461,Y 0.112,Z -325.930,A 0.00099,B 0.00000,C 180.00000} ; release
  LIN {X 14079.461,Y 0.112,Z -25.930,A 0.00099,B 0.00000,C 180.00000} ; retreat
  ; Step 775, bar 1088
  LIN {X -14079.461,Y 0.112,Z 868.364,A 179.99901,B 0.00000,C -180.00000} ; outside
  LIN {X -14079.461,Y 0.112,Z -75.930,A 179.99901,B 0.00000,C -180.00000} ; preinsert
  LIN {X -14079.461,Y 0.112,Z -325.930,A 179.99901,B 0.00000,C -180.00000} ; insert
  LIN {X -14079.461,Y 0.112,Z -325.930,A 179.99901,B 0.00000,C -180.00000} ; release
  LIN {X -14079.461,Y 0.112,Z -25.930,A 179.99901,B 0.00000,C -180.00000} ; retreat
  ; Step 776, bar 1098
  LIN {X -14079.461,Y 149.888,Z 868.364,A -179.99901,B 0.00000,C -180.00000} ; outside
  LIN {X -14079.461,Y 149.888,Z -75.930,A -179.99901,B 0.00000,C -180.00000} ; preinsert
  LIN {X -14079.461,Y 149.888,Z -325.930,A -179.99901,B 0.00000,C -180.00000} ; insert
  LIN {X -14079.461,Y 149.888,Z -325.930,A -179.99901,B 0.00000,C -180.00000} ; release
  LIN {X -14079.461,Y 149.888,Z -25.930,A -179.99901,B 0.00000,C -180.00000} ; retreat
  ; Step 777, bar 1077
  LIN {X 14079.461,Y 149.888,Z 868.364,A -0.00099,B 0.00000,C 180.00000} ; outside
  LIN {X 14079.461,Y 149.888,Z -75.930,A -0.00099,B 0.00000,C 180.00000} ; preinsert
  LIN {X 14079.461,Y 149.888,Z -325.930,A -0.00099,B 0.00000,C 180.00000} ; insert
  LIN {X 14079.461,Y 149.888,Z -325.930,A -0.00099,B 0.00000,C 180.00000} ; release
  LIN {X 14079.461,Y 149.888,Z -25.930,A -0.00099,B 0.00000,C 180.00000} ; retreat
  ; Step 778, bar 1099
  LIN {X -14079.461,Y 299.888,Z 868.364,A -179.99901,B 0.00000,C -180.00000} ; outside
  LIN {X -14079.461,Y 299.888,Z -75.930,A -179.99901,B 0.00000,C -180.00000} ; preinsert
  LIN {X -14079.461,Y 299.888,Z -325.930,A -179.99901,B 0.00000,C -180.00000} ; insert
  LIN {X -14079.461,Y 299.888,Z -325.930,A -179.99901,B 0.00000,C -180.00000} ; release
  LIN {X -14079.461,Y 299.888,Z -25.930,A -179.99901,B 0.00000,C -180.00000} ; retreat
  ; Step 779, bar 1078
  LIN {X 14079.461,Y 299.888,Z 868.364,A -0.00099,B 0.00000,C 180.00000} ; outside
  LIN {X 14079.461,Y 299.888,Z -75.930,A -0.00099,B 0.00000,C 180.00000} ; preinsert
  LIN {X 14079.461,Y 299.888,Z -325.930,A -0.00099,B 0.00000,C 180.00000} ; insert
  LIN {X 14079.461,Y 299.888,Z -325.930,A -0.00099,B 0.00000,C 180.00000} ; release
  LIN {X 14079.461,Y 299.888,Z -25.930,A -0.00099,B 0.00000,C 180.00000} ; retreat
  ; Step 780, bar 1100
  LIN {X -14079.461,Y 449.888,Z 868.364,A -179.99901,B 0.00000,C -180.00000} ; outside
  LIN {X -14079.461,Y 449.888,Z -75.930,A -179.99901,B 0.00000,C -180.00000} ; preinsert
  LIN {X -14079.461,Y 449.888,Z -325.930,A -179.99901,B 0.00000,C -180.00000} ; insert
  LIN {X -14079.461,Y 449.888,Z -325.930,A -179.99901,B 0.00000,C -180.00000} ; release
  LIN {X -14079.461,Y 449.888,Z -25.930,A -179.99901,B 0.00000,C -180.00000} ; retreat
  ; Step 781, bar 1079
  LIN {X 14079.461,Y 449.888,Z 868.364,A -0.00099,B 0.00000,C 180.00000} ; outside
  LIN {X 14079.461,Y 449.888,Z -75.930,A -0.00099,B 0.00000,C 180.00000} ; preinsert
  LIN {X 14079.461,Y 449.888,Z -325.930,A -0.00099,B 0.00000,C 180.00000} ; insert
  LIN {X 14079.461,Y 449.888,Z -325.930,A -0.00099,B 0.00000,C 180.00000} ; release
  LIN {X 14079.461,Y 449.888,Z -25.930,A -0.00099,B 0.00000,C 180.00000} ; retreat
  ; Step 782, bar 1101
  LIN {X -14079.461,Y 599.888,Z 868.364,A -179.99901,B 0.00000,C 180.00000} ; outside
  LIN {X -14079.461,Y 599.888,Z -75.930,A -179.99901,B 0.00000,C 180.00000} ; preinsert
  LIN {X -14079.461,Y 599.888,Z -325.930,A -179.99901,B 0.00000,C 180.00000} ; insert
  LIN {X -14079.461,Y 599.888,Z -325.930,A -179.99901,B 0.00000,C 180.00000} ; release
  LIN {X -14079.461,Y 599.888,Z -25.930,A -179.99901,B 0.00000,C 180.00000} ; retreat
  ; Step 783, bar 1080
  LIN {X 14079.461,Y 599.888,Z 868.364,A -0.00099,B 0.00000,C 180.00000} ; outside
  LIN {X 14079.461,Y 599.888,Z -75.930,A -0.00099,B 0.00000,C 180.00000} ; preinsert
  LIN {X 14079.461,Y 599.888,Z -325.930,A -0.00099,B 0.00000,C 180.00000} ; insert
  LIN {X 14079.461,Y 599.888,Z -325.930,A -0.00099,B 0.00000,C 180.00000} ; release
  LIN {X 14079.461,Y 599.888,Z -25.930,A -0.00099,B 0.00000,C 180.00000} ; retreat
  ; Step 784, bar 1102
  LIN {X -14079.461,Y 749.888,Z 868.364,A -179.99901,B 0.00000,C 180.00000} ; outside
  LIN {X -14079.461,Y 749.888,Z -75.930,A -179.99901,B 0.00000,C 180.00000} ; preinsert
  LIN {X -14079.461,Y 749.888,Z -325.930,A -179.99901,B 0.00000,C 180.00000} ; insert
  LIN {X -14079.461,Y 749.888,Z -325.930,A -179.99901,B 0.00000,C 180.00000} ; release
  LIN {X -14079.461,Y 749.888,Z -25.930,A -179.99901,B 0.00000,C 180.00000} ; retreat
  ; Step 785, bar 1081
  LIN {X 14079.461,Y 749.888,Z 868.364,A -0.00099,B 0.00000,C 180.00000} ; outside
  LIN {X 14079.461,Y 749.888,Z -75.930,A -0.00099,B 0.00000,C 180.00000} ; preinsert
  LIN {X 14079.461,Y 749.888,Z -325.930,A -0.00099,B 0.00000,C 180.00000} ; insert
  LIN {X 14079.461,Y 749.888,Z -325.930,A -0.00099,B 0.00000,C 180.00000} ; release
  LIN {X 14079.461,Y 749.888,Z -25.930,A -0.00099,B 0.00000,C 180.00000} ; retreat
  ; Step 786, bar 1103
  LIN {X -14079.461,Y 899.888,Z 868.364,A -179.99901,B 0.00000,C 180.00000} ; outside
  LIN {X -14079.461,Y 899.888,Z -75.930,A -179.99901,B 0.00000,C 180.00000} ; preinsert
  LIN {X -14079.461,Y 899.888,Z -325.930,A -179.99901,B 0.00000,C 180.00000} ; insert
  LIN {X -14079.461,Y 899.888,Z -325.930,A -179.99901,B 0.00000,C 180.00000} ; release
  LIN {X -14079.461,Y 899.888,Z -25.930,A -179.99901,B 0.00000,C 180.00000} ; retreat
  ; Step 787, bar 1082
  LIN {X 14079.461,Y 899.888,Z 868.364,A -0.00099,B 0.00000,C 180.00000} ; outside
  LIN {X 14079.461,Y 899.888,Z -75.930,A -0.00099,B 0.00000,C 180.00000} ; preinsert
  LIN {X 14079.461,Y 899.888,Z -325.930,A -0.00099,B 0.00000,C 180.00000} ; insert
  LIN {X 14079.461,Y 899.888,Z -325.930,A -0.00099,B 0.00000,C 180.00000} ; release
  LIN {X 14079.461,Y 899.888,Z -25.930,A -0.00099,B 0.00000,C 180.00000} ; retreat
  ; Step 788, bar 1104
  LIN {X -14079.461,Y 1049.888,Z 868.364,A -179.99901,B 0.00000,C -180.00000} ; outside
  LIN {X -14079.461,Y 1049.888,Z -75.930,A -179.99901,B 0.00000,C -180.00000} ; preinsert
  LIN {X -14079.461,Y 1049.888,Z -325.930,A -179.99901,B 0.00000,C -180.00000} ; insert
  LIN {X -14079.461,Y 1049.888,Z -325.930,A -179.99901,B 0.00000,C -180.00000} ; release
  LIN {X -14079.461,Y 1049.888,Z -25.930,A -179.99901,B 0.00000,C -180.00000} ; retreat
  ; Step 789, bar 1083
  LIN {X 14079.461,Y 1049.888,Z 868.364,A -0.00099,B 0.00000,C 180.00000} ; outside
  LIN {X 14079.461,Y 1049.888,Z -75.930,A -0.00099,B 0.00000,C 180.00000} ; preinsert
  LIN {X 14079.461,Y 1049.888,Z -325.930,A -0.00099,B 0.00000,C 180.00000} ; insert
  LIN {X 14079.461,Y 1049.888,Z -325.930,A -0.00099,B 0.00000,C 180.00000} ; release
  LIN {X 14079.461,Y 1049.888,Z -25.930,A -0.00099,B 0.00000,C 180.00000} ; retreat
  ; Step 790, bar 1105
  LIN {X -14079.461,Y 1374.888,Z 868.364,A -179.99901,B 0.00000,C -180.00000} ; outside
  LIN {X -14079.461,Y 1374.888,Z -75.930,A -179.99901,B 0.00000,C -180.00000} ; preinsert
  LIN {X -14079.461,Y 1374.888,Z -325.930,A -179.99901,B 0.00000,C -180.00000} ; insert
  LIN {X -14079.461,Y 1374.888,Z -325.930,A -179.99901,B 0.00000,C -180.00000} ; release
  LIN {X -14079.461,Y 1374.888,Z -25.930,A -179.99901,B 0.00000,C -180.00000} ; retreat
  ; Step 791, bar 1086
  LIN {X 14079.461,Y 1374.888,Z 868.364,A -0.00099,B 0.00000,C 180.00000} ; outside
  LIN {X 14079.461,Y 1374.888,Z -75.930,A -0.00099,B 0.00000,C 180.00000} ; preinsert
  LIN {X 14079.461,Y 1374.888,Z -325.930,A -0.00099,B 0.00000,C 180.00000} ; insert
  LIN {X 14079.461,Y 1374.888,Z -325.930,A -0.00099,B 0.00000,C 180.00000} ; release
  LIN {X 14079.461,Y 1374.888,Z -25.930,A -0.00099,B 0.00000,C 180.00000} ; retreat
  ; Step 792, bar 1106
  LIN {X -14079.461,Y 1499.888,Z 868.364,A -179.99901,B 0.00000,C -180.00000} ; outside
  LIN {X -14079.461,Y 1499.888,Z -75.930,A -179.99901,B 0.00000,C -180.00000} ; preinsert
  LIN {X -14079.461,Y 1499.888,Z -325.930,A -179.99901,B 0.00000,C -180.00000} ; insert
  LIN {X -14079.461,Y 1499.888,Z -325.930,A -179.99901,B 0.00000,C -180.00000} ; release
  LIN {X -14079.461,Y 1499.888,Z -25.930,A -179.99901,B 0.00000,C -180.00000} ; retreat
  ; Step 793, bar 1087
  LIN {X 14079.461,Y 1499.888,Z 868.364,A -0.00099,B 0.00000,C 180.00000} ; outside
  LIN {X 14079.461,Y 1499.888,Z -75.930,A -0.00099,B 0.00000,C 180.00000} ; preinsert
  LIN {X 14079.461,Y 1499.888,Z -325.930,A -0.00099,B 0.00000,C 180.00000} ; insert
  LIN {X 14079.461,Y 1499.888,Z -325.930,A -0.00099,B 0.00000,C 180.00000} ; release
  LIN {X 14079.461,Y 1499.888,Z -25.930,A -0.00099,B 0.00000,C 180.00000} ; retreat
  ; Step 794, bar 289
  LIN {X 0.000,Y -1420.000,Z 1081.871,A 0.00000,B 0.00000,C 180.00000} ; outside
  LIN {X 0.000,Y -1420.000,Z 165.246,A 0.00000,B 0.00000,C 180.00000} ; preinsert
  LIN {X 0.000,Y -1420.000,Z -84.754,A 0.00000,B 0.00000,C 180.00000} ; insert
  LIN {X 0.000,Y -1420.000,Z -84.754,A 0.00000,B 0.00000,C 180.00000} ; release
  LIN {X 0.000,Y -1420.000,Z 215.246,A 0.00000,B 0.00000,C 180.00000} ; retreat
  ; Step 795, bar 316
  LIN {X 0.000,Y 1420.000,Z 1081.871,A 0.00000,B 0.00000,C 180.00000} ; outside
  LIN {X 0.000,Y 1420.000,Z 165.246,A 0.00000,B 0.00000,C 180.00000} ; preinsert
  LIN {X 0.000,Y 1420.000,Z -84.754,A 0.00000,B 0.00000,C 180.00000} ; insert
  LIN {X 0.000,Y 1420.000,Z -84.754,A 0.00000,B 0.00000,C 180.00000} ; release
  LIN {X 0.000,Y 1420.000,Z 215.246,A 0.00000,B 0.00000,C 180.00000} ; retreat
  ; Step 796, bar 288
  LIN {X 0.000,Y -1325.000,Z 1085.621,A 0.00000,B 0.00000,C 180.00000} ; outside
  LIN {X 0.000,Y -1325.000,Z 167.121,A 0.00000,B 0.00000,C 180.00000} ; preinsert
  LIN {X 0.000,Y -1325.000,Z -82.879,A 0.00000,B 0.00000,C 180.00000} ; insert
  LIN {X 0.000,Y -1325.000,Z -82.879,A 0.00000,B 0.00000,C 180.00000} ; release
  LIN {X 0.000,Y -1325.000,Z 217.121,A 0.00000,B 0.00000,C 180.00000} ; retreat
  ; Step 797, bar 315
  LIN {X 0.000,Y 1325.000,Z 1085.621,A 0.00000,B 0.00000,C 180.00000} ; outside
  LIN {X 0.000,Y 1325.000,Z 167.121,A 0.00000,B 0.00000,C 180.00000} ; preinsert
  LIN {X 0.000,Y 1325.000,Z -82.879,A 0.00000,B 0.00000,C 180.00000} ; insert
  LIN {X 0.000,Y 1325.000,Z -82.879,A 0.00000,B 0.00000,C 180.00000} ; release
  LIN {X 0.000,Y 1325.000,Z 217.121,A 0.00000,B 0.00000,C 180.00000} ; retreat
  ; Step 798, bar 3107
  LIN {X -15204.133,Y -1216.217,Z 1079.276,A -179.87076,B 0.00000,C -180.00000} ; outside
  LIN {X -15204.133,Y -1216.217,Z 93.267,A -179.87076,B 0.00000,C -180.00000} ; preinsert
  LIN {X -15204.133,Y -1216.217,Z -156.733,A -179.87076,B 0.00000,C -180.00000} ; insert
  LIN {X -15204.133,Y -1216.217,Z -156.733,A -179.87076,B 0.00000,C -180.00000} ; release
  LIN {X -15204.133,Y -1216.217,Z 143.267,A -179.87076,B 0.00000,C -180.00000} ; retreat
  ; Step 799, bar 3097
  LIN {X 15204.133,Y -1216.217,Z 1079.276,A -0.12924,B 0.00000,C 180.00000} ; outside
  LIN {X 15204.133,Y -1216.217,Z 93.267,A -0.12924,B 0.00000,C 180.00000} ; preinsert
  LIN {X 15204.133,Y -1216.217,Z -156.733,A -0.12924,B 0.00000,C 180.00000} ; insert
  LIN {X 15204.133,Y -1216.217,Z -156.733,A -0.12924,B 0.00000,C 180.00000} ; release
  LIN {X 15204.133,Y -1216.217,Z 143.267,A -0.12924,B 0.00000,C 180.00000} ; retreat
  ; Step 800, bar 3102
  LIN {X -15204.133,Y 1216.217,Z 1079.276,A 179.87076,B 0.00000,C -180.00000} ; outside
  LIN {X -15204.133,Y 1216.217,Z 93.267,A 179.87076,B 0.00000,C -180.00000} ; preinsert
  LIN {X -15204.133,Y 1216.217,Z -156.733,A 179.87076,B 0.00000,C -180.00000} ; insert
  LIN {X -15204.133,Y 1216.217,Z -156.733,A 179.87076,B 0.00000,C -180.00000} ; release
  LIN {X -15204.133,Y 1216.217,Z 143.267,A 179.87076,B 0.00000,C -180.00000} ; retreat
  ; Step 801, bar 3092
  LIN {X 15204.133,Y 1216.217,Z 1079.276,A 0.12924,B 0.00000,C 180.00000} ; outside
  LIN {X 15204.133,Y 1216.217,Z 93.267,A 0.12924,B 0.00000,C 180.00000} ; preinsert
  LIN {X 15204.133,Y 1216.217,Z -156.733,A 0.12924,B 0.00000,C 180.00000} ; insert
  LIN {X 15204.133,Y 1216.217,Z -156.733,A 0.12924,B 0.00000,C 180.00000} ; release
  LIN {X 15204.133,Y 1216.217,Z 143.267,A 0.12924,B 0.00000,C 180.00000} ; retreat
  ; Step 802, bar 287
  LIN {X 0.000,Y -1200.000,Z 1090.621,A 0.00000,B 0.00000,C 180.00000} ; outside
  LIN {X 0.000,Y -1200.000,Z 169.621,A 0.00000,B 0.00000,C 180.00000} ; preinsert
  LIN {X 0.000,Y -1200.000,Z -80.379,A 0.00000,B 0.00000,C 180.00000} ; insert
  LIN {X 0.000,Y -1200.000,Z -80.379,A 0.00000,B 0.00000,C 180.00000} ; release
  LIN {X 0.000,Y -1200.000,Z 219.621,A 0.00000,B 0.00000,C 180.00000} ; retreat
  ; Step 803, bar 314
  LIN {X 0.000,Y 1200.000,Z 1090.621,A 0.00000,B 0.00000,C 180.00000} ; outside
  LIN {X 0.000,Y 1200.000,Z 169.621,A 0.00000,B 0.00000,C 180.00000} ; preinsert
  LIN {X 0.000,Y 1200.000,Z -80.379,A 0.00000,B 0.00000,C 180.00000} ; insert
  LIN {X 0.000,Y 1200.000,Z -80.379,A 0.00000,B 0.00000,C 180.00000} ; release
  LIN {X 0.000,Y 1200.000,Z 219.621,A 0.00000,B 0.00000,C 180.00000} ; retreat
  ; Step 804, bar 286
  LIN {X -0.147,Y -1049.934,Z 1096.488,A -179.99973,B 0.00000,C -180.00000} ; outside
  LIN {X -0.147,Y -1049.934,Z 172.549,A -179.99973,B 0.00000,C -180.00000} ; preinsert
  LIN {X -0.147,Y -1049.934,Z -77.451,A -179.99973,B 0.00000,C -180.00000} ; insert
  LIN {X -0.147,Y -1049.934,Z -77.451,A -179.99973,B 0.00000,C -180.00000} ; release
  LIN {X -0.147,Y -1049.934,Z 222.549,A -179.99973,B 0.00000,C -180.00000} ; retreat
  ; Step 805, bar 313
  LIN {X -0.146,Y 1049.934,Z 1096.488,A 179.99973,B 0.00000,C 180.00000} ; outside
  LIN {X -0.146,Y 1049.934,Z 172.549,A 179.99973,B 0.00000,C 180.00000} ; preinsert
  LIN {X -0.146,Y 1049.934,Z -77.451,A 179.99973,B 0.00000,C 180.00000} ; insert
  LIN {X -0.146,Y 1049.934,Z -77.451,A 179.99973,B 0.00000,C 180.00000} ; release
  LIN {X -0.146,Y 1049.934,Z 222.549,A 179.99973,B 0.00000,C 180.00000} ; retreat
  ; Step 806, bar 3106
  LIN {X -15204.133,Y -891.217,Z 1079.276,A -179.87076,B 0.00000,C 180.00000} ; outside
  LIN {X -15204.133,Y -891.217,Z 98.892,A -179.87076,B 0.00000,C 180.00000} ; preinsert
  LIN {X -15204.133,Y -891.217,Z -151.108,A -179.87076,B 0.00000,C 180.00000} ; insert
  LIN {X -15204.133,Y -891.217,Z -151.108,A -179.87076,B 0.00000,C 180.00000} ; release
  LIN {X -15204.133,Y -891.217,Z 148.892,A -179.87076,B 0.00000,C 180.00000} ; retreat
  ; Step 807, bar 3096
  LIN {X 15204.133,Y -891.217,Z 1079.276,A -0.12924,B 0.00000,C 180.00000} ; outside
  LIN {X 15204.133,Y -891.217,Z 98.892,A -0.12924,B 0.00000,C 180.00000} ; preinsert
  LIN {X 15204.133,Y -891.217,Z -151.108,A -0.12924,B 0.00000,C 180.00000} ; insert
  LIN {X 15204.133,Y -891.217,Z -151.108,A -0.12924,B 0.00000,C 180.00000} ; release
  LIN {X 15204.133,Y -891.217,Z 148.892,A -0.12924,B 0.00000,C 180.00000} ; retreat
  ; Step 808, bar 3101
  LIN {X -15204.133,Y 891.217,Z 1079.276,A 179.87076,B 0.00000,C 180.00000} ; outside
  LIN {X -15204.133,Y 891.217,Z 98.892,A 179.87076,B 0.00000,C 180.00000} ; preinsert
  LIN {X -15204.133,Y 891.217,Z -151.108,A 179.87076,B 0.00000,C 180.00000} ; insert
  LIN {X -15204.133,Y 891.217,Z -151.108,A 179.87076,B 0.00000,C 180.00000} ; release
  LIN {X -15204.133,Y 891.217,Z 148.892,A 179.87076,B 0.00000,C 180.00000} ; retreat
  ; Step 809, bar 3091
  LIN {X 15204.133,Y 891.217,Z 1079.276,A 0.12924,B 0.00000,C 180.00000} ; outside
  LIN {X 15204.133,Y 891.217,Z 98.892,A 0.12924,B 0.00000,C 180.00000} ; preinsert
  LIN {X 15204.133,Y 891.217,Z -151.108,A 0.12924,B 0.00000,C 180.00000} ; insert
  LIN {X 15204.133,Y 891.217,Z -151.108,A 0.12924,B 0.00000,C 180.00000} ; release
  LIN {X 15204.133,Y 891.217,Z 148.892,A 0.12924,B 0.00000,C 180.00000} ; retreat
  ; Step 810, bar 1887
  LIN {X -15947.499,Y -1050.009,Z 1097.463,A 179.99947,B 0.00000,C 180.00000} ; outside
  LIN {X -15947.499,Y -1050.009,Z 173.034,A 179.99947,B 0.00000,C 180.00000} ; preinsert
  LIN {X -15947.499,Y -1050.009,Z -76.966,A 179.99947,B 0.00000,C 180.00000} ; insert
  LIN {X -15947.499,Y -1050.009,Z -76.966,A 179.99947,B 0.00000,C 180.00000} ; release
  LIN {X -15947.499,Y -1050.009,Z 223.034,A 179.99947,B 0.00000,C 180.00000} ; retreat
  ; Step 811, bar 1891
  LIN {X 15947.499,Y -1050.009,Z 1097.463,A 0.00053,B 0.00000,C 180.00000} ; outside
  LIN {X 15947.499,Y -1050.009,Z 173.034,A 0.00053,B 0.00000,C 180.00000} ; preinsert
  LIN {X 15947.499,Y -1050.009,Z -76.966,A 0.00053,B 0.00000,C 180.00000} ; insert
  LIN {X 15947.499,Y -1050.009,Z -76.966,A 0.00053,B 0.00000,C 180.00000} ; release
  LIN {X 15947.499,Y -1050.009,Z 223.034,A 0.00053,B 0.00000,C 180.00000} ; retreat
  ; Step 812, bar 1885
  LIN {X -15052.602,Y -1049.764,Z 1097.832,A 179.98657,B 0.00000,C -180.00000} ; outside
  LIN {X -15052.602,Y -1049.764,Z 173.210,A 179.98657,B 0.00000,C -180.00000} ; preinsert
  LIN {X -15052.602,Y -1049.764,Z -76.790,A 179.98657,B 0.00000,C -180.00000} ; insert
  LIN {X -15052.602,Y -1049.764,Z -76.790,A 179.98657,B 0.00000,C -180.00000} ; release
  LIN {X -15052.602,Y -1049.764,Z 223.210,A 179.98657,B 0.00000,C -180.00000} ; retreat
  ; Step 813, bar 1889
  LIN {X 15052.602,Y -1049.764,Z 1097.832,A 0.01343,B 0.00000,C 180.00000} ; outside
  LIN {X 15052.602,Y -1049.764,Z 173.210,A 0.01343,B 0.00000,C 180.00000} ; preinsert
  LIN {X 15052.602,Y -1049.764,Z -76.790,A 0.01343,B 0.00000,C 180.00000} ; insert
  LIN {X 15052.602,Y -1049.764,Z -76.790,A 0.01343,B 0.00000,C 180.00000} ; release
  LIN {X 15052.602,Y -1049.764,Z 223.210,A 0.01343,B 0.00000,C 180.00000} ; retreat
  ; Step 814, bar 1886
  LIN {X -15052.602,Y 1049.764,Z 1097.832,A -179.98657,B 0.00000,C -180.00000} ; outside
  LIN {X -15052.602,Y 1049.764,Z 173.210,A -179.98657,B 0.00000,C -180.00000} ; preinsert
  LIN {X -15052.602,Y 1049.764,Z -76.790,A -179.98657,B 0.00000,C -180.00000} ; insert
  LIN {X -15052.602,Y 1049.764,Z -76.790,A -179.98657,B 0.00000,C -180.00000} ; release
  LIN {X -15052.602,Y 1049.764,Z 223.210,A -179.98657,B 0.00000,C -180.00000} ; retreat
  ; Step 815, bar 1890
  LIN {X 15052.602,Y 1049.764,Z 1097.832,A -0.01343,B 0.00000,C 180.00000} ; outside
  LIN {X 15052.602,Y 1049.764,Z 173.210,A -0.01343,B 0.00000,C 180.00000} ; preinsert
  LIN {X 15052.602,Y 1049.764,Z -76.790,A -0.01343,B 0.00000,C 180.00000} ; insert
  LIN {X 15052.602,Y 1049.764,Z -76.790,A -0.01343,B 0.00000,C 180.00000} ; release
  LIN {X 15052.602,Y 1049.764,Z 223.210,A -0.01343,B 0.00000,C 180.00000} ; retreat
  ; Step 816, bar 1888
  LIN {X -15947.499,Y 1050.009,Z 1097.463,A -179.99947,B 0.00000,C -180.00000} ; outside
  LIN {X -15947.499,Y 1050.009,Z 173.034,A -179.99947,B 0.00000,C -180.00000} ; preinsert
  LIN {X -15947.499,Y 1050.009,Z -76.966,A -179.99947,B 0.00000,C -180.00000} ; insert
  LIN {X -15947.499,Y 1050.009,Z -76.966,A -179.99947,B 0.00000,C -180.00000} ; release
  LIN {X -15947.499,Y 1050.009,Z 223.034,A -179.99947,B 0.00000,C -180.00000} ; retreat
  ; Step 817, bar 1892
  LIN {X 15947.499,Y 1050.009,Z 1097.463,A -0.00053,B 0.00000,C 180.00000} ; outside
  LIN {X 15947.499,Y 1050.009,Z 173.034,A -0.00053,B 0.00000,C 180.00000} ; preinsert
  LIN {X 15947.499,Y 1050.009,Z -76.966,A -0.00053,B 0.00000,C 180.00000} ; insert
  LIN {X 15947.499,Y 1050.009,Z -76.966,A -0.00053,B 0.00000,C 180.00000} ; release
  LIN {X 15947.499,Y 1050.009,Z 223.034,A -0.00053,B 0.00000,C 180.00000} ; retreat
  ; Step 818, bar 304
  LIN {X 0.000,Y -3490.000,Z 1099.371,A 0.00000,B 0.00000,C 180.00000} ; outside
  LIN {X 0.000,Y -3490.000,Z 173.996,A 0.00000,B 0.00000,C 180.00000} ; preinsert
  LIN {X 0.000,Y -3490.000,Z -76.004,A 0.00000,B 0.00000,C 180.00000} ; insert
  LIN {X 0.000,Y -3490.000,Z -76.004,A 0.00000,B 0.00000,C 180.00000} ; release
  LIN {X 0.000,Y -3490.000,Z 223.996,A 0.00000,B 0.00000,C 180.00000} ; retreat
  ; Step 819, bar 331
  LIN {X 0.000,Y 3490.000,Z 1099.371,A 0.00000,B 0.00000,C 180.00000} ; outside
  LIN {X 0.000,Y 3490.000,Z 173.996,A 0.00000,B 0.00000,C 180.00000} ; preinsert
  LIN {X 0.000,Y 3490.000,Z -76.004,A 0.00000,B 0.00000,C 180.00000} ; insert
  LIN {X 0.000,Y 3490.000,Z -76.004,A 0.00000,B 0.00000,C 180.00000} ; release
  LIN {X 0.000,Y 3490.000,Z 223.996,A 0.00000,B 0.00000,C 180.00000} ; retreat
  ; Step 820, bar 285
  LIN {X 0.000,Y -875.000,Z 1101.871,A 0.00000,B 0.00000,C 180.00000} ; outside
  LIN {X 0.000,Y -875.000,Z 175.246,A 0.00000,B 0.00000,C 180.00000} ; preinsert
  LIN {X 0.000,Y -875.000,Z -74.754,A 0.00000,B 0.00000,C 180.00000} ; insert
  LIN {X 0.000,Y -875.000,Z -74.754,A 0.00000,B 0.00000,C 180.00000} ; release
  LIN {X 0.000,Y -875.000,Z 225.246,A 0.00000,B 0.00000,C 180.00000} ; retreat
  ; Step 821, bar 312
  LIN {X 0.000,Y 875.000,Z 1101.871,A 0.00000,B 0.00000,C 180.00000} ; outside
  LIN {X 0.000,Y 875.000,Z 175.246,A 0.00000,B 0.00000,C 180.00000} ; preinsert
  LIN {X 0.000,Y 875.000,Z -74.754,A 0.00000,B 0.00000,C 180.00000} ; insert
  LIN {X 0.000,Y 875.000,Z -74.754,A 0.00000,B 0.00000,C 180.00000} ; release
  LIN {X 0.000,Y 875.000,Z 225.246,A 0.00000,B 0.00000,C 180.00000} ; retreat
  ; Step 822, bar 2392
  LIN {X 375.007,Y -1961.237,Z 950.053,A -87.94718,B 0.00000,C 180.00000} ; outside
  LIN {X 375.007,Y -1961.237,Z 18.185,A -87.94718,B 0.00000,C 180.00000} ; preinsert
  LIN {X 375.007,Y -1961.237,Z -231.815,A -87.94718,B 0.00000,C 180.00000} ; insert
  LIN {X 375.007,Y -1961.237,Z -231.815,A -87.94718,B 0.00000,C 180.00000} ; release
  LIN {X 375.007,Y -1961.237,Z 68.185,A -87.94718,B 0.00000,C 180.00000} ; retreat
  ; Step 823, bar 2398
  LIN {X 1125.007,Y -1961.237,Z 950.053,A -87.94718,B 0.00000,C 180.00000} ; outside
  LIN {X 1125.007,Y -1961.237,Z 18.185,A -87.94718,B 0.00000,C 180.00000} ; preinsert
  LIN {X 1125.007,Y -1961.237,Z -231.815,A -87.94718,B 0.00000,C 180.00000} ; insert
  LIN {X 1125.007,Y -1961.237,Z -231.815,A -87.94718,B 0.00000,C 180.00000} ; release
  LIN {X 1125.007,Y -1961.237,Z 68.185,A -87.94718,B 0.00000,C 180.00000} ; retreat
  ; Step 824, bar 2404
  LIN {X 1875.007,Y -1961.237,Z 950.053,A -87.94718,B 0.00000,C 180.00000} ; outside
  LIN {X 1875.007,Y -1961.237,Z 18.185,A -87.94718,B 0.00000,C 180.00000} ; preinsert
  LIN {X 1875.007,Y -1961.237,Z -231.815,A -87.94718,B 0.00000,C 180.00000} ; insert
  LIN {X 1875.007,Y -1961.237,Z -231.815,A -87.94718,B 0.00000,C 180.00000} ; release
  LIN {X 1875.007,Y -1961.237,Z 68.185,A -87.94718,B 0.00000,C 180.00000} ; retreat
  ; Step 825, bar 2410
  LIN {X 2625.007,Y -1961.237,Z 950.053,A -87.94718,B 0.00000,C 180.00000} ; outside
  LIN {X 2625.007,Y -1961.237,Z 18.185,A -87.94718,B 0.00000,C 180.00000} ; preinsert
  LIN {X 2625.007,Y -1961.237,Z -231.815,A -87.94718,B 0.00000,C 180.00000} ; insert
  LIN {X 2625.007,Y -1961.237,Z -231.815,A -87.94718,B 0.00000,C 180.00000} ; release
  LIN {X 2625.007,Y -1961.237,Z 68.185,A -87.94718,B 0.00000,C 180.00000} ; retreat
  ; Step 826, bar 2416
  LIN {X 3375.007,Y -1961.237,Z 950.053,A -87.94718,B 0.00000,C 180.00000} ; outside
  LIN {X 3375.007,Y -1961.237,Z 18.185,A -87.94718,B 0.00000,C 180.00000} ; preinsert
  LIN {X 3375.007,Y -1961.237,Z -231.815,A -87.94718,B 0.00000,C 180.00000} ; insert
  LIN {X 3375.007,Y -1961.237,Z -231.815,A -87.94718,B 0.00000,C 180.00000} ; release
  LIN {X 3375.007,Y -1961.237,Z 68.185,A -87.94718,B 0.00000,C 180.00000} ; retreat
  ; Step 827, bar 2422
  LIN {X 4125.007,Y -1961.237,Z 950.053,A -87.94718,B 0.00000,C 180.00000} ; outside
  LIN {X 4125.007,Y -1961.237,Z 18.185,A -87.94718,B 0.00000,C 180.00000} ; preinsert
  LIN {X 4125.007,Y -1961.237,Z -231.815,A -87.94718,B 0.00000,C 180.00000} ; insert
  LIN {X 4125.007,Y -1961.237,Z -231.815,A -87.94718,B 0.00000,C 180.00000} ; release
  LIN {X 4125.007,Y -1961.237,Z 68.185,A -87.94718,B 0.00000,C 180.00000} ; retreat
  ; Step 828, bar 2428
  LIN {X 4875.007,Y -1961.237,Z 950.053,A -87.94718,B 0.00000,C 180.00000} ; outside
  LIN {X 4875.007,Y -1961.237,Z 18.185,A -87.94718,B 0.00000,C 180.00000} ; preinsert
  LIN {X 4875.007,Y -1961.237,Z -231.815,A -87.94718,B 0.00000,C 180.00000} ; insert
  LIN {X 4875.007,Y -1961.237,Z -231.815,A -87.94718,B 0.00000,C 180.00000} ; release
  LIN {X 4875.007,Y -1961.237,Z 68.185,A -87.94718,B 0.00000,C 180.00000} ; retreat
  ; Step 829, bar 2434
  LIN {X 5625.007,Y -1961.237,Z 950.053,A -87.94718,B 0.00000,C 180.00000} ; outside
  LIN {X 5625.007,Y -1961.237,Z 18.185,A -87.94718,B 0.00000,C 180.00000} ; preinsert
  LIN {X 5625.007,Y -1961.237,Z -231.815,A -87.94718,B 0.00000,C 180.00000} ; insert
  LIN {X 5625.007,Y -1961.237,Z -231.815,A -87.94718,B 0.00000,C 180.00000} ; release
  LIN {X 5625.007,Y -1961.237,Z 68.185,A -87.94718,B 0.00000,C 180.00000} ; retreat
  ; Step 830, bar 2440
  LIN {X 6375.007,Y -1961.237,Z 950.053,A -87.94718,B 0.00000,C 180.00000} ; outside
  LIN {X 6375.007,Y -1961.237,Z 18.185,A -87.94718,B 0.00000,C 180.00000} ; preinsert
  LIN {X 6375.007,Y -1961.237,Z -231.815,A -87.94718,B 0.00000,C 180.00000} ; insert
  LIN {X 6375.007,Y -1961.237,Z -231.815,A -87.94718,B 0.00000,C 180.00000} ; release
  LIN {X 6375.007,Y -1961.237,Z 68.185,A -87.94718,B 0.00000,C 180.00000} ; retreat
  ; Step 831, bar 2446
  LIN {X 7125.007,Y -1961.237,Z 950.053,A -87.94718,B 0.00000,C 180.00000} ; outside
  LIN {X 7125.007,Y -1961.237,Z 18.185,A -87.94718,B 0.00000,C 180.00000} ; preinsert
  LIN {X 7125.007,Y -1961.237,Z -231.815,A -87.94718,B 0.00000,C 180.00000} ; insert
  LIN {X 7125.007,Y -1961.237,Z -231.815,A -87.94718,B 0.00000,C 180.00000} ; release
  LIN {X 7125.007,Y -1961.237,Z 68.185,A -87.94718,B 0.00000,C 180.00000} ; retreat
  ; Step 832, bar 2452
  LIN {X 7875.007,Y -1961.237,Z 950.053,A -87.94718,B 0.00000,C 180.00000} ; outside
  LIN {X 7875.007,Y -1961.237,Z 18.185,A -87.94718,B 0.00000,C 180.00000} ; preinsert
  LIN {X 7875.007,Y -1961.237,Z -231.815,A -87.94718,B 0.00000,C 180.00000} ; insert
  LIN {X 7875.007,Y -1961.237,Z -231.815,A -87.94718,B 0.00000,C 180.00000} ; release
  LIN {X 7875.007,Y -1961.237,Z 68.185,A -87.94718,B 0.00000,C 180.00000} ; retreat
  ; Step 833, bar 2458
  LIN {X 8625.007,Y -1961.237,Z 950.053,A -87.94718,B 0.00000,C 180.00000} ; outside
  LIN {X 8625.007,Y -1961.237,Z 18.185,A -87.94718,B 0.00000,C 180.00000} ; preinsert
  LIN {X 8625.007,Y -1961.237,Z -231.815,A -87.94718,B 0.00000,C 180.00000} ; insert
  LIN {X 8625.007,Y -1961.237,Z -231.815,A -87.94718,B 0.00000,C 180.00000} ; release
  LIN {X 8625.007,Y -1961.237,Z 68.185,A -87.94718,B 0.00000,C 180.00000} ; retreat
  ; Step 834, bar 2464
  LIN {X 9375.007,Y -1961.237,Z 950.053,A -87.94718,B 0.00000,C 180.00000} ; outside
  LIN {X 9375.007,Y -1961.237,Z 18.185,A -87.94718,B 0.00000,C 180.00000} ; preinsert
  LIN {X 9375.007,Y -1961.237,Z -231.815,A -87.94718,B 0.00000,C 180.00000} ; insert
  LIN {X 9375.007,Y -1961.237,Z -231.815,A -87.94718,B 0.00000,C 180.00000} ; release
  LIN {X 9375.007,Y -1961.237,Z 68.185,A -87.94718,B 0.00000,C 180.00000} ; retreat
  ; Step 835, bar 2470
  LIN {X 10125.007,Y -1961.237,Z 950.053,A -87.94718,B 0.00000,C 180.00000} ; outside
  LIN {X 10125.007,Y -1961.237,Z 18.185,A -87.94718,B 0.00000,C 180.00000} ; preinsert
  LIN {X 10125.007,Y -1961.237,Z -231.815,A -87.94718,B 0.00000,C 180.00000} ; insert
  LIN {X 10125.007,Y -1961.237,Z -231.815,A -87.94718,B 0.00000,C 180.00000} ; release
  LIN {X 10125.007,Y -1961.237,Z 68.185,A -87.94718,B 0.00000,C 180.00000} ; retreat
  ; Step 836, bar 2476
  LIN {X 10875.007,Y -1961.237,Z 950.053,A -87.94718,B 0.00000,C 180.00000} ; outside
  LIN {X 10875.007,Y -1961.237,Z 18.185,A -87.94718,B 0.00000,C 180.00000} ; preinsert
  LIN {X 10875.007,Y -1961.237,Z -231.815,A -87.94718,B 0.00000,C 180.00000} ; insert
  LIN {X 10875.007,Y -1961.237,Z -231.815,A -87.94718,B 0.00000,C 180.00000} ; release
  LIN {X 10875.007,Y -1961.237,Z 68.185,A -87.94718,B 0.00000,C 180.00000} ; retreat
  ; Step 837, bar 2482
  LIN {X 11625.007,Y -1961.237,Z 950.053,A -87.94718,B 0.00000,C 180.00000} ; outside
  LIN {X 11625.007,Y -1961.237,Z 18.185,A -87.94718,B 0.00000,C 180.00000} ; preinsert
  LIN {X 11625.007,Y -1961.237,Z -231.815,A -87.94718,B 0.00000,C 180.00000} ; insert
  LIN {X 11625.007,Y -1961.237,Z -231.815,A -87.94718,B 0.00000,C 180.00000} ; release
  LIN {X 11625.007,Y -1961.237,Z 68.185,A -87.94718,B 0.00000,C 180.00000} ; retreat
  ; Step 838, bar 2488
  LIN {X 12250.007,Y -1961.237,Z 950.053,A -87.94718,B 0.00000,C 180.00000} ; outside
  LIN {X 12250.007,Y -1961.237,Z 18.185,A -87.94718,B 0.00000,C 180.00000} ; preinsert
  LIN {X 12250.007,Y -1961.237,Z -231.815,A -87.94718,B 0.00000,C 180.00000} ; insert
  LIN {X 12250.007,Y -1961.237,Z -231.815,A -87.94718,B 0.00000,C 180.00000} ; release
  LIN {X 12250.007,Y -1961.237,Z 68.185,A -87.94718,B 0.00000,C 180.00000} ; retreat
  ; Step 839, bar 2494
  LIN {X 12850.007,Y -1961.237,Z 950.053,A -87.94718,B 0.00000,C 180.00000} ; outside
  LIN {X 12850.007,Y -1961.237,Z 18.185,A -87.94718,B 0.00000,C 180.00000} ; preinsert
  LIN {X 12850.007,Y -1961.237,Z -231.815,A -87.94718,B 0.00000,C 180.00000} ; insert
  LIN {X 12850.007,Y -1961.237,Z -231.815,A -87.94718,B 0.00000,C 180.00000} ; release
  LIN {X 12850.007,Y -1961.237,Z 68.185,A -87.94718,B 0.00000,C 180.00000} ; retreat
  ; Step 840, bar 2500
  LIN {X 13450.007,Y -1961.237,Z 950.053,A -87.94718,B 0.00000,C 180.00000} ; outside
  LIN {X 13450.007,Y -1961.237,Z 18.185,A -87.94718,B 0.00000,C 180.00000} ; preinsert
  LIN {X 13450.007,Y -1961.237,Z -231.815,A -87.94718,B 0.00000,C 180.00000} ; insert
  LIN {X 13450.007,Y -1961.237,Z -231.815,A -87.94718,B 0.00000,C 180.00000} ; release
  LIN {X 13450.007,Y -1961.237,Z 68.185,A -87.94718,B 0.00000,C 180.00000} ; retreat
  ; Step 841, bar 2506
  LIN {X 14050.007,Y -1961.237,Z 950.053,A -87.94718,B 0.00000,C 180.00000} ; outside
  LIN {X 14050.007,Y -1961.237,Z 18.185,A -87.94718,B 0.00000,C 180.00000} ; preinsert
  LIN {X 14050.007,Y -1961.237,Z -231.815,A -87.94718,B 0.00000,C 180.00000} ; insert
  LIN {X 14050.007,Y -1961.237,Z -231.815,A -87.94718,B 0.00000,C 180.00000} ; release
  LIN {X 14050.007,Y -1961.237,Z 68.185,A -87.94718,B 0.00000,C 180.00000} ; retreat
  ; Step 842, bar 2512
  LIN {X 14650.007,Y -1961.237,Z 950.053,A -87.94718,B 0.00000,C 180.00000} ; outside
  LIN {X 14650.007,Y -1961.237,Z 18.185,A -87.94718,B 0.00000,C 180.00000} ; preinsert
  LIN {X 14650.007,Y -1961.237,Z -231.815,A -87.94718,B 0.00000,C 180.00000} ; insert
  LIN {X 14650.007,Y -1961.237,Z -231.815,A -87.94718,B 0.00000,C 180.00000} ; release
  LIN {X 14650.007,Y -1961.237,Z 68.185,A -87.94718,B 0.00000,C 180.00000} ; retreat
  ; Step 843, bar 2518
  LIN {X 15250.007,Y -1961.237,Z 950.053,A -87.94718,B 0.00000,C 180.00000} ; outside
  LIN {X 15250.007,Y -1961.237,Z 18.185,A -87.94718,B 0.00000,C 180.00000} ; preinsert
  LIN {X 15250.007,Y -1961.237,Z -231.815,A -87.94718,B 0.00000,C 180.00000} ; insert
  LIN {X 15250.007,Y -1961.237,Z -231.815,A -87.94718,B 0.00000,C 180.00000} ; release
  LIN {X 15250.007,Y -1961.237,Z 68.185,A -87.94718,B 0.00000,C 180.00000} ; retreat
  ; Step 844, bar 2524
  LIN {X 15850.007,Y -1961.237,Z 950.053,A -87.94718,B 0.00000,C 180.00000} ; outside
  LIN {X 15850.007,Y -1961.237,Z 18.185,A -87.94718,B 0.00000,C 180.00000} ; preinsert
  LIN {X 15850.007,Y -1961.237,Z -231.815,A -87.94718,B 0.00000,C 180.00000} ; insert
  LIN {X 15850.007,Y -1961.237,Z -231.815,A -87.94718,B 0.00000,C 180.00000} ; release
  LIN {X 15850.007,Y -1961.237,Z 68.185,A -87.94718,B 0.00000,C 180.00000} ; retreat
  ; Step 845, bar 2107
  LIN {X -15850.007,Y 1961.237,Z 950.053,A 92.05282,B 0.00000,C 180.00000} ; outside
  LIN {X -15850.007,Y 1961.237,Z 18.185,A 92.05282,B 0.00000,C 180.00000} ; preinsert
  LIN {X -15850.007,Y 1961.237,Z -231.815,A 92.05282,B 0.00000,C 180.00000} ; insert
  LIN {X -15850.007,Y 1961.237,Z -231.815,A 92.05282,B 0.00000,C 180.00000} ; release
  LIN {X -15850.007,Y 1961.237,Z 68.185,A 92.05282,B 0.00000,C 180.00000} ; retreat
  ; Step 846, bar 2101
  LIN {X -15250.007,Y 1961.237,Z 950.053,A 92.05282,B 0.00000,C 180.00000} ; outside
  LIN {X -15250.007,Y 1961.237,Z 18.185,A 92.05282,B 0.00000,C 180.00000} ; preinsert
  LIN {X -15250.007,Y 1961.237,Z -231.815,A 92.05282,B 0.00000,C 180.00000} ; insert
  LIN {X -15250.007,Y 1961.237,Z -231.815,A 92.05282,B 0.00000,C 180.00000} ; release
  LIN {X -15250.007,Y 1961.237,Z 68.185,A 92.05282,B 0.00000,C 180.00000} ; retreat
  ; Step 847, bar 2095
  LIN {X -14650.007,Y 1961.237,Z 950.053,A 92.05282,B 0.00000,C 180.00000} ; outside
  LIN {X -14650.007,Y 1961.237,Z 18.185,A 92.05282,B 0.00000,C 180.00000} ; preinsert
  LIN {X -14650.007,Y 1961.237,Z -231.815,A 92.05282,B 0.00000,C 180.00000} ; insert
  LIN {X -14650.007,Y 1961.237,Z -231.815,A 92.05282,B 0.00000,C 180.00000} ; release
  LIN {X -14650.007,Y 1961.237,Z 68.185,A 92.05282,B 0.00000,C 180.00000} ; retreat
  ; Step 848, bar 2089
  LIN {X -14050.007,Y 1961.237,Z 950.053,A 92.05282,B 0.00000,C 180.00000} ; outside
  LIN {X -14050.007,Y 1961.237,Z 18.185,A 92.05282,B 0.00000,C 180.00000} ; preinsert
  LIN {X -14050.007,Y 1961.237,Z -231.815,A 92.05282,B 0.00000,C 180.00000} ; insert
  LIN {X -14050.007,Y 1961.237,Z -231.815,A 92.05282,B 0.00000,C 180.00000} ; release
  LIN {X -14050.007,Y 1961.237,Z 68.185,A 92.05282,B 0.00000,C 180.00000} ; retreat
  ; Step 849, bar 2083
  LIN {X -13450.007,Y 1961.237,Z 950.053,A 92.05282,B 0.00000,C 180.00000} ; outside
  LIN {X -13450.007,Y 1961.237,Z 18.185,A 92.05282,B 0.00000,C 180.00000} ; preinsert
  LIN {X -13450.007,Y 1961.237,Z -231.815,A 92.05282,B 0.00000,C 180.00000} ; insert
  LIN {X -13450.007,Y 1961.237,Z -231.815,A 92.05282,B 0.00000,C 180.00000} ; release
  LIN {X -13450.007,Y 1961.237,Z 68.185,A 92.05282,B 0.00000,C 180.00000} ; retreat
  ; Step 850, bar 2077
  LIN {X -12850.007,Y 1961.237,Z 950.053,A 92.05282,B 0.00000,C 180.00000} ; outside
  LIN {X -12850.007,Y 1961.237,Z 18.185,A 92.05282,B 0.00000,C 180.00000} ; preinsert
  LIN {X -12850.007,Y 1961.237,Z -231.815,A 92.05282,B 0.00000,C 180.00000} ; insert
  LIN {X -12850.007,Y 1961.237,Z -231.815,A 92.05282,B 0.00000,C 180.00000} ; release
  LIN {X -12850.007,Y 1961.237,Z 68.185,A 92.05282,B 0.00000,C 180.00000} ; retreat
  ; Step 851, bar 2071
  LIN {X -12250.007,Y 1961.237,Z 950.053,A 92.05282,B 0.00000,C 180.00000} ; outside
  LIN {X -12250.007,Y 1961.237,Z 18.185,A 92.05282,B 0.00000,C 180.00000} ; preinsert
  LIN {X -12250.007,Y 1961.237,Z -231.815,A 92.05282,B 0.00000,C 180.00000} ; insert
  LIN {X -12250.007,Y 1961.237,Z -231.815,A 92.05282,B 0.00000,C 180.00000} ; release
  LIN {X -12250.007,Y 1961.237,Z 68.185,A 92.05282,B 0.00000,C 180.00000} ; retreat
  ; Step 852, bar 2065
  LIN {X -11625.007,Y 1961.237,Z 950.053,A 92.05282,B 0.00000,C 180.00000} ; outside
  LIN {X -11625.007,Y 1961.237,Z 18.185,A 92.05282,B 0.00000,C 180.00000} ; preinsert
  LIN {X -11625.007,Y 1961.237,Z -231.815,A 92.05282,B 0.00000,C 180.00000} ; insert
  LIN {X -11625.007,Y 1961.237,Z -231.815,A 92.05282,B 0.00000,C 180.00000} ; release
  LIN {X -11625.007,Y 1961.237,Z 68.185,A 92.05282,B 0.00000,C 180.00000} ; retreat
  ; Step 853, bar 2059
  LIN {X -10875.007,Y 1961.237,Z 950.053,A 92.05282,B 0.00000,C 180.00000} ; outside
  LIN {X -10875.007,Y 1961.237,Z 18.185,A 92.05282,B 0.00000,C 180.00000} ; preinsert
  LIN {X -10875.007,Y 1961.237,Z -231.815,A 92.05282,B 0.00000,C 180.00000} ; insert
  LIN {X -10875.007,Y 1961.237,Z -231.815,A 92.05282,B 0.00000,C 180.00000} ; release
  LIN {X -10875.007,Y 1961.237,Z 68.185,A 92.05282,B 0.00000,C 180.00000} ; retreat
  ; Step 854, bar 2053
  LIN {X -10125.007,Y 1961.237,Z 950.053,A 92.05282,B 0.00000,C 180.00000} ; outside
  LIN {X -10125.007,Y 1961.237,Z 18.185,A 92.05282,B 0.00000,C 180.00000} ; preinsert
  LIN {X -10125.007,Y 1961.237,Z -231.815,A 92.05282,B 0.00000,C 180.00000} ; insert
  LIN {X -10125.007,Y 1961.237,Z -231.815,A 92.05282,B 0.00000,C 180.00000} ; release
  LIN {X -10125.007,Y 1961.237,Z 68.185,A 92.05282,B 0.00000,C 180.00000} ; retreat
  ; Step 855, bar 2047
  LIN {X -9375.007,Y 1961.237,Z 950.053,A 92.05282,B 0.00000,C 180.00000} ; outside
  LIN {X -9375.007,Y 1961.237,Z 18.185,A 92.05282,B 0.00000,C 180.00000} ; preinsert
  LIN {X -9375.007,Y 1961.237,Z -231.815,A 92.05282,B 0.00000,C 180.00000} ; insert
  LIN {X -9375.007,Y 1961.237,Z -231.815,A 92.05282,B 0.00000,C 180.00000} ; release
  LIN {X -9375.007,Y 1961.237,Z 68.185,A 92.05282,B 0.00000,C 180.00000} ; retreat
  ; Step 856, bar 2041
  LIN {X -8625.007,Y 1961.237,Z 950.053,A 92.05282,B 0.00000,C 180.00000} ; outside
  LIN {X -8625.007,Y 1961.237,Z 18.185,A 92.05282,B 0.00000,C 180.00000} ; preinsert
  LIN {X -8625.007,Y 1961.237,Z -231.815,A 92.05282,B 0.00000,C 180.00000} ; insert
  LIN {X -8625.007,Y 1961.237,Z -231.815,A 92.05282,B 0.00000,C 180.00000} ; release
  LIN {X -8625.007,Y 1961.237,Z 68.185,A 92.05282,B 0.00000,C 180.00000} ; retreat
  ; Step 857, bar 2035
  LIN {X -7875.007,Y 1961.237,Z 950.053,A 92.05282,B 0.00000,C -180.00000} ; outside
  LIN {X -7875.007,Y 1961.237,Z 18.185,A 92.05282,B 0.00000,C -180.00000} ; preinsert
  LIN {X -7875.007,Y 1961.237,Z -231.815,A 92.05282,B 0.00000,C -180.00000} ; insert
  LIN {X -7875.007,Y 1961.237,Z -231.815,A 92.05282,B 0.00000,C -180.00000} ; release
  LIN {X -7875.007,Y 1961.237,Z 68.185,A 92.05282,B 0.00000,C -180.00000} ; retreat
  ; Step 858, bar 2029
  LIN {X -7125.007,Y 1961.237,Z 950.053,A 92.05282,B 0.00000,C -180.00000} ; outside
  LIN {X -7125.007,Y 1961.237,Z 18.185,A 92.05282,B 0.00000,C -180.00000} ; preinsert
  LIN {X -7125.007,Y 1961.237,Z -231.815,A 92.05282,B 0.00000,C -180.00000} ; insert
  LIN {X -7125.007,Y 1961.237,Z -231.815,A 92.05282,B 0.00000,C -180.00000} ; release
  LIN {X -7125.007,Y 1961.237,Z 68.185,A 92.05282,B 0.00000,C -180.00000} ; retreat
  ; Step 859, bar 2023
  LIN {X -6375.007,Y 1961.237,Z 950.053,A 92.05282,B 0.00000,C -180.00000} ; outside
  LIN {X -6375.007,Y 1961.237,Z 18.185,A 92.05282,B 0.00000,C -180.00000} ; preinsert
  LIN {X -6375.007,Y 1961.237,Z -231.815,A 92.05282,B 0.00000,C -180.00000} ; insert
  LIN {X -6375.007,Y 1961.237,Z -231.815,A 92.05282,B 0.00000,C -180.00000} ; release
  LIN {X -6375.007,Y 1961.237,Z 68.185,A 92.05282,B 0.00000,C -180.00000} ; retreat
  ; Step 860, bar 2017
  LIN {X -5625.007,Y 1961.237,Z 950.053,A 92.05282,B 0.00000,C -180.00000} ; outside
  LIN {X -5625.007,Y 1961.237,Z 18.185,A 92.05282,B 0.00000,C -180.00000} ; preinsert
  LIN {X -5625.007,Y 1961.237,Z -231.815,A 92.05282,B 0.00000,C -180.00000} ; insert
  LIN {X -5625.007,Y 1961.237,Z -231.815,A 92.05282,B 0.00000,C -180.00000} ; release
  LIN {X -5625.007,Y 1961.237,Z 68.185,A 92.05282,B 0.00000,C -180.00000} ; retreat
  ; Step 861, bar 2011
  LIN {X -4875.007,Y 1961.237,Z 950.053,A 92.05282,B 0.00000,C -180.00000} ; outside
  LIN {X -4875.007,Y 1961.237,Z 18.185,A 92.05282,B 0.00000,C -180.00000} ; preinsert
  LIN {X -4875.007,Y 1961.237,Z -231.815,A 92.05282,B 0.00000,C -180.00000} ; insert
  LIN {X -4875.007,Y 1961.237,Z -231.815,A 92.05282,B 0.00000,C -180.00000} ; release
  LIN {X -4875.007,Y 1961.237,Z 68.185,A 92.05282,B 0.00000,C -180.00000} ; retreat
  ; Step 862, bar 2005
  LIN {X -4125.007,Y 1961.237,Z 950.053,A 92.05282,B 0.00000,C -180.00000} ; outside
  LIN {X -4125.007,Y 1961.237,Z 18.185,A 92.05282,B 0.00000,C -180.00000} ; preinsert
  LIN {X -4125.007,Y 1961.237,Z -231.815,A 92.05282,B 0.00000,C -180.00000} ; insert
  LIN {X -4125.007,Y 1961.237,Z -231.815,A 92.05282,B 0.00000,C -180.00000} ; release
  LIN {X -4125.007,Y 1961.237,Z 68.185,A 92.05282,B 0.00000,C -180.00000} ; retreat
  ; Step 863, bar 1999
  LIN {X -3375.007,Y 1961.237,Z 950.053,A 92.05282,B 0.00000,C -180.00000} ; outside
  LIN {X -3375.007,Y 1961.237,Z 18.185,A 92.05282,B 0.00000,C -180.00000} ; preinsert
  LIN {X -3375.007,Y 1961.237,Z -231.815,A 92.05282,B 0.00000,C -180.00000} ; insert
  LIN {X -3375.007,Y 1961.237,Z -231.815,A 92.05282,B 0.00000,C -180.00000} ; release
  LIN {X -3375.007,Y 1961.237,Z 68.185,A 92.05282,B 0.00000,C -180.00000} ; retreat
  ; Step 864, bar 1993
  LIN {X -2625.007,Y 1961.237,Z 950.053,A 92.05282,B 0.00000,C -180.00000} ; outside
  LIN {X -2625.007,Y 1961.237,Z 18.185,A 92.05282,B 0.00000,C -180.00000} ; preinsert
  LIN {X -2625.007,Y 1961.237,Z -231.815,A 92.05282,B 0.00000,C -180.00000} ; insert
  LIN {X -2625.007,Y 1961.237,Z -231.815,A 92.05282,B 0.00000,C -180.00000} ; release
  LIN {X -2625.007,Y 1961.237,Z 68.185,A 92.05282,B 0.00000,C -180.00000} ; retreat
  ; Step 865, bar 1987
  LIN {X -1875.007,Y 1961.237,Z 950.053,A 92.05282,B 0.00000,C -180.00000} ; outside
  LIN {X -1875.007,Y 1961.237,Z 18.185,A 92.05282,B 0.00000,C -180.00000} ; preinsert
  LIN {X -1875.007,Y 1961.237,Z -231.815,A 92.05282,B 0.00000,C -180.00000} ; insert
  LIN {X -1875.007,Y 1961.237,Z -231.815,A 92.05282,B 0.00000,C -180.00000} ; release
  LIN {X -1875.007,Y 1961.237,Z 68.185,A 92.05282,B 0.00000,C -180.00000} ; retreat
  ; Step 866, bar 1981
  LIN {X -1125.007,Y 1961.237,Z 950.053,A 92.05282,B 0.00000,C -180.00000} ; outside
  LIN {X -1125.007,Y 1961.237,Z 18.185,A 92.05282,B 0.00000,C -180.00000} ; preinsert
  LIN {X -1125.007,Y 1961.237,Z -231.815,A 92.05282,B 0.00000,C -180.00000} ; insert
  LIN {X -1125.007,Y 1961.237,Z -231.815,A 92.05282,B 0.00000,C -180.00000} ; release
  LIN {X -1125.007,Y 1961.237,Z 68.185,A 92.05282,B 0.00000,C -180.00000} ; retreat
  ; Step 867, bar 1968
  LIN {X -375.007,Y 1961.237,Z 950.053,A 92.05282,B 0.00000,C 180.00000} ; outside
  LIN {X -375.007,Y 1961.237,Z 18.185,A 92.05282,B 0.00000,C 180.00000} ; preinsert
  LIN {X -375.007,Y 1961.237,Z -231.815,A 92.05282,B 0.00000,C 180.00000} ; insert
  LIN {X -375.007,Y 1961.237,Z -231.815,A 92.05282,B 0.00000,C 180.00000} ; release
  LIN {X -375.007,Y 1961.237,Z 68.185,A 92.05282,B 0.00000,C 180.00000} ; retreat
  ; Step 868, bar 2386
  LIN {X -15850.007,Y -1961.237,Z 950.053,A -92.05282,B 0.00000,C -180.00000} ; outside
  LIN {X -15850.007,Y -1961.237,Z 18.185,A -92.05282,B 0.00000,C -180.00000} ; preinsert
  LIN {X -15850.007,Y -1961.237,Z -231.815,A -92.05282,B 0.00000,C -180.00000} ; insert
  LIN {X -15850.007,Y -1961.237,Z -231.815,A -92.05282,B 0.00000,C -180.00000} ; release
  LIN {X -15850.007,Y -1961.237,Z 68.185,A -92.05282,B 0.00000,C -180.00000} ; retreat
  ; Step 869, bar 2380
  LIN {X -15250.007,Y -1961.237,Z 950.053,A -92.05282,B 0.00000,C -180.00000} ; outside
  LIN {X -15250.007,Y -1961.237,Z 18.185,A -92.05282,B 0.00000,C -180.00000} ; preinsert
  LIN {X -15250.007,Y -1961.237,Z -231.815,A -92.05282,B 0.00000,C -180.00000} ; insert
  LIN {X -15250.007,Y -1961.237,Z -231.815,A -92.05282,B 0.00000,C -180.00000} ; release
  LIN {X -15250.007,Y -1961.237,Z 68.185,A -92.05282,B 0.00000,C -180.00000} ; retreat
  ; Step 870, bar 2374
  LIN {X -14650.007,Y -1961.237,Z 950.053,A -92.05282,B 0.00000,C -180.00000} ; outside
  LIN {X -14650.007,Y -1961.237,Z 18.185,A -92.05282,B 0.00000,C -180.00000} ; preinsert
  LIN {X -14650.007,Y -1961.237,Z -231.815,A -92.05282,B 0.00000,C -180.00000} ; insert
  LIN {X -14650.007,Y -1961.237,Z -231.815,A -92.05282,B 0.00000,C -180.00000} ; release
  LIN {X -14650.007,Y -1961.237,Z 68.185,A -92.05282,B 0.00000,C -180.00000} ; retreat
  ; Step 871, bar 2368
  LIN {X -14050.007,Y -1961.237,Z 950.053,A -92.05282,B 0.00000,C -180.00000} ; outside
  LIN {X -14050.007,Y -1961.237,Z 18.185,A -92.05282,B 0.00000,C -180.00000} ; preinsert
  LIN {X -14050.007,Y -1961.237,Z -231.815,A -92.05282,B 0.00000,C -180.00000} ; insert
  LIN {X -14050.007,Y -1961.237,Z -231.815,A -92.05282,B 0.00000,C -180.00000} ; release
  LIN {X -14050.007,Y -1961.237,Z 68.185,A -92.05282,B 0.00000,C -180.00000} ; retreat
  ; Step 872, bar 2362
  LIN {X -13450.007,Y -1961.237,Z 950.053,A -92.05282,B 0.00000,C -180.00000} ; outside
  LIN {X -13450.007,Y -1961.237,Z 18.185,A -92.05282,B 0.00000,C -180.00000} ; preinsert
  LIN {X -13450.007,Y -1961.237,Z -231.815,A -92.05282,B 0.00000,C -180.00000} ; insert
  LIN {X -13450.007,Y -1961.237,Z -231.815,A -92.05282,B 0.00000,C -180.00000} ; release
  LIN {X -13450.007,Y -1961.237,Z 68.185,A -92.05282,B 0.00000,C -180.00000} ; retreat
  ; Step 873, bar 2356
  LIN {X -12850.007,Y -1961.237,Z 950.053,A -92.05282,B 0.00000,C -180.00000} ; outside
  LIN {X -12850.007,Y -1961.237,Z 18.185,A -92.05282,B 0.00000,C -180.00000} ; preinsert
  LIN {X -12850.007,Y -1961.237,Z -231.815,A -92.05282,B 0.00000,C -180.00000} ; insert
  LIN {X -12850.007,Y -1961.237,Z -231.815,A -92.05282,B 0.00000,C -180.00000} ; release
  LIN {X -12850.007,Y -1961.237,Z 68.185,A -92.05282,B 0.00000,C -180.00000} ; retreat
  ; Step 874, bar 2350
  LIN {X -12250.007,Y -1961.237,Z 950.053,A -92.05282,B 0.00000,C -180.00000} ; outside
  LIN {X -12250.007,Y -1961.237,Z 18.185,A -92.05282,B 0.00000,C -180.00000} ; preinsert
  LIN {X -12250.007,Y -1961.237,Z -231.815,A -92.05282,B 0.00000,C -180.00000} ; insert
  LIN {X -12250.007,Y -1961.237,Z -231.815,A -92.05282,B 0.00000,C -180.00000} ; release
  LIN {X -12250.007,Y -1961.237,Z 68.185,A -92.05282,B 0.00000,C -180.00000} ; retreat
  ; Step 875, bar 2344
  LIN {X -11625.007,Y -1961.237,Z 950.053,A -92.05282,B 0.00000,C -180.00000} ; outside
  LIN {X -11625.007,Y -1961.237,Z 18.185,A -92.05282,B 0.00000,C -180.00000} ; preinsert
  LIN {X -11625.007,Y -1961.237,Z -231.815,A -92.05282,B 0.00000,C -180.00000} ; insert
  LIN {X -11625.007,Y -1961.237,Z -231.815,A -92.05282,B 0.00000,C -180.00000} ; release
  LIN {X -11625.007,Y -1961.237,Z 68.185,A -92.05282,B 0.00000,C -180.00000} ; retreat
  ; Step 876, bar 2338
  LIN {X -10875.007,Y -1961.237,Z 950.053,A -92.05282,B 0.00000,C -180.00000} ; outside
  LIN {X -10875.007,Y -1961.237,Z 18.185,A -92.05282,B 0.00000,C -180.00000} ; preinsert
  LIN {X -10875.007,Y -1961.237,Z -231.815,A -92.05282,B 0.00000,C -180.00000} ; insert
  LIN {X -10875.007,Y -1961.237,Z -231.815,A -92.05282,B 0.00000,C -180.00000} ; release
  LIN {X -10875.007,Y -1961.237,Z 68.185,A -92.05282,B 0.00000,C -180.00000} ; retreat
  ; Step 877, bar 2332
  LIN {X -10125.007,Y -1961.237,Z 950.053,A -92.05282,B 0.00000,C -180.00000} ; outside
  LIN {X -10125.007,Y -1961.237,Z 18.185,A -92.05282,B 0.00000,C -180.00000} ; preinsert
  LIN {X -10125.007,Y -1961.237,Z -231.815,A -92.05282,B 0.00000,C -180.00000} ; insert
  LIN {X -10125.007,Y -1961.237,Z -231.815,A -92.05282,B 0.00000,C -180.00000} ; release
  LIN {X -10125.007,Y -1961.237,Z 68.185,A -92.05282,B 0.00000,C -180.00000} ; retreat
  ; Step 878, bar 2326
  LIN {X -9375.007,Y -1961.237,Z 950.053,A -92.05282,B 0.00000,C -180.00000} ; outside
  LIN {X -9375.007,Y -1961.237,Z 18.185,A -92.05282,B 0.00000,C -180.00000} ; preinsert
  LIN {X -9375.007,Y -1961.237,Z -231.815,A -92.05282,B 0.00000,C -180.00000} ; insert
  LIN {X -9375.007,Y -1961.237,Z -231.815,A -92.05282,B 0.00000,C -180.00000} ; release
  LIN {X -9375.007,Y -1961.237,Z 68.185,A -92.05282,B 0.00000,C -180.00000} ; retreat
  ; Step 879, bar 2320
  LIN {X -8625.007,Y -1961.237,Z 950.053,A -92.05282,B 0.00000,C -180.00000} ; outside
  LIN {X -8625.007,Y -1961.237,Z 18.185,A -92.05282,B 0.00000,C -180.00000} ; preinsert
  LIN {X -8625.007,Y -1961.237,Z -231.815,A -92.05282,B 0.00000,C -180.00000} ; insert
  LIN {X -8625.007,Y -1961.237,Z -231.815,A -92.05282,B 0.00000,C -180.00000} ; release
  LIN {X -8625.007,Y -1961.237,Z 68.185,A -92.05282,B 0.00000,C -180.00000} ; retreat
  ; Step 880, bar 2314
  LIN {X -7875.007,Y -1961.237,Z 950.053,A -92.05282,B 0.00000,C 180.00000} ; outside
  LIN {X -7875.007,Y -1961.237,Z 18.185,A -92.05282,B 0.00000,C 180.00000} ; preinsert
  LIN {X -7875.007,Y -1961.237,Z -231.815,A -92.05282,B 0.00000,C 180.00000} ; insert
  LIN {X -7875.007,Y -1961.237,Z -231.815,A -92.05282,B 0.00000,C 180.00000} ; release
  LIN {X -7875.007,Y -1961.237,Z 68.185,A -92.05282,B 0.00000,C 180.00000} ; retreat
  ; Step 881, bar 2308
  LIN {X -7125.007,Y -1961.237,Z 950.053,A -92.05282,B 0.00000,C 180.00000} ; outside
  LIN {X -7125.007,Y -1961.237,Z 18.185,A -92.05282,B 0.00000,C 180.00000} ; preinsert
  LIN {X -7125.007,Y -1961.237,Z -231.815,A -92.05282,B 0.00000,C 180.00000} ; insert
  LIN {X -7125.007,Y -1961.237,Z -231.815,A -92.05282,B 0.00000,C 180.00000} ; release
  LIN {X -7125.007,Y -1961.237,Z 68.185,A -92.05282,B 0.00000,C 180.00000} ; retreat
  ; Step 882, bar 2302
  LIN {X -6375.007,Y -1961.237,Z 950.053,A -92.05282,B 0.00000,C 180.00000} ; outside
  LIN {X -6375.007,Y -1961.237,Z 18.185,A -92.05282,B 0.00000,C 180.00000} ; preinsert
  LIN {X -6375.007,Y -1961.237,Z -231.815,A -92.05282,B 0.00000,C 180.00000} ; insert
  LIN {X -6375.007,Y -1961.237,Z -231.815,A -92.05282,B 0.00000,C 180.00000} ; release
  LIN {X -6375.007,Y -1961.237,Z 68.185,A -92.05282,B 0.00000,C 180.00000} ; retreat
  ; Step 883, bar 2296
  LIN {X -5625.007,Y -1961.237,Z 950.053,A -92.05282,B 0.00000,C 180.00000} ; outside
  LIN {X -5625.007,Y -1961.237,Z 18.185,A -92.05282,B 0.00000,C 180.00000} ; preinsert
  LIN {X -5625.007,Y -1961.237,Z -231.815,A -92.05282,B 0.00000,C 180.00000} ; insert
  LIN {X -5625.007,Y -1961.237,Z -231.815,A -92.05282,B 0.00000,C 180.00000} ; release
  LIN {X -5625.007,Y -1961.237,Z 68.185,A -92.05282,B 0.00000,C 180.00000} ; retreat
  ; Step 884, bar 2290
  LIN {X -4875.007,Y -1961.237,Z 950.053,A -92.05282,B 0.00000,C 180.00000} ; outside
  LIN {X -4875.007,Y -1961.237,Z 18.185,A -92.05282,B 0.00000,C 180.00000} ; preinsert
  LIN {X -4875.007,Y -1961.237,Z -231.815,A -92.05282,B 0.00000,C 180.00000} ; insert
  LIN {X -4875.007,Y -1961.237,Z -231.815,A -92.05282,B 0.00000,C 180.00000} ; release
  LIN {X -4875.007,Y -1961.237,Z 68.185,A -92.05282,B 0.00000,C 180.00000} ; retreat
  ; Step 885, bar 2284
  LIN {X -4125.007,Y -1961.237,Z 950.053,A -92.05282,B 0.00000,C 180.00000} ; outside
  LIN {X -4125.007,Y -1961.237,Z 18.185,A -92.05282,B 0.00000,C 180.00000} ; preinsert
  LIN {X -4125.007,Y -1961.237,Z -231.815,A -92.05282,B 0.00000,C 180.00000} ; insert
  LIN {X -4125.007,Y -1961.237,Z -231.815,A -92.05282,B 0.00000,C 180.00000} ; release
  LIN {X -4125.007,Y -1961.237,Z 68.185,A -92.05282,B 0.00000,C 180.00000} ; retreat
  ; Step 886, bar 2278
  LIN {X -3375.007,Y -1961.237,Z 950.053,A -92.05282,B 0.00000,C 180.00000} ; outside
  LIN {X -3375.007,Y -1961.237,Z 18.185,A -92.05282,B 0.00000,C 180.00000} ; preinsert
  LIN {X -3375.007,Y -1961.237,Z -231.815,A -92.05282,B 0.00000,C 180.00000} ; insert
  LIN {X -3375.007,Y -1961.237,Z -231.815,A -92.05282,B 0.00000,C 180.00000} ; release
  LIN {X -3375.007,Y -1961.237,Z 68.185,A -92.05282,B 0.00000,C 180.00000} ; retreat
  ; Step 887, bar 2272
  LIN {X -2625.007,Y -1961.237,Z 950.053,A -92.05282,B 0.00000,C 180.00000} ; outside
  LIN {X -2625.007,Y -1961.237,Z 18.185,A -92.05282,B 0.00000,C 180.00000} ; preinsert
  LIN {X -2625.007,Y -1961.237,Z -231.815,A -92.05282,B 0.00000,C 180.00000} ; insert
  LIN {X -2625.007,Y -1961.237,Z -231.815,A -92.05282,B 0.00000,C 180.00000} ; release
  LIN {X -2625.007,Y -1961.237,Z 68.185,A -92.05282,B 0.00000,C 180.00000} ; retreat
  ; Step 888, bar 2266
  LIN {X -1875.007,Y -1961.237,Z 950.053,A -92.05282,B 0.00000,C 180.00000} ; outside
  LIN {X -1875.007,Y -1961.237,Z 18.185,A -92.05282,B 0.00000,C 180.00000} ; preinsert
  LIN {X -1875.007,Y -1961.237,Z -231.815,A -92.05282,B 0.00000,C 180.00000} ; insert
  LIN {X -1875.007,Y -1961.237,Z -231.815,A -92.05282,B 0.00000,C 180.00000} ; release
  LIN {X -1875.007,Y -1961.237,Z 68.185,A -92.05282,B 0.00000,C 180.00000} ; retreat
  ; Step 889, bar 2260
  LIN {X -1125.007,Y -1961.237,Z 950.053,A -92.05282,B 0.00000,C 180.00000} ; outside
  LIN {X -1125.007,Y -1961.237,Z 18.185,A -92.05282,B 0.00000,C 180.00000} ; preinsert
  LIN {X -1125.007,Y -1961.237,Z -231.815,A -92.05282,B 0.00000,C 180.00000} ; insert
  LIN {X -1125.007,Y -1961.237,Z -231.815,A -92.05282,B 0.00000,C 180.00000} ; release
  LIN {X -1125.007,Y -1961.237,Z 68.185,A -92.05282,B 0.00000,C 180.00000} ; retreat
  ; Step 890, bar 2254
  LIN {X -375.007,Y -1961.237,Z 950.053,A -92.05282,B 0.00000,C -180.00000} ; outside
  LIN {X -375.007,Y -1961.237,Z 18.185,A -92.05282,B 0.00000,C -180.00000} ; preinsert
  LIN {X -375.007,Y -1961.237,Z -231.815,A -92.05282,B 0.00000,C -180.00000} ; insert
  LIN {X -375.007,Y -1961.237,Z -231.815,A -92.05282,B 0.00000,C -180.00000} ; release
  LIN {X -375.007,Y -1961.237,Z 68.185,A -92.05282,B 0.00000,C -180.00000} ; retreat
  ; Step 891, bar 2113
  LIN {X 375.007,Y 1961.237,Z 950.053,A 87.94718,B 0.00000,C 180.00000} ; outside
  LIN {X 375.007,Y 1961.237,Z 18.185,A 87.94718,B 0.00000,C 180.00000} ; preinsert
  LIN {X 375.007,Y 1961.237,Z -231.815,A 87.94718,B 0.00000,C 180.00000} ; insert
  LIN {X 375.007,Y 1961.237,Z -231.815,A 87.94718,B 0.00000,C 180.00000} ; release
  LIN {X 375.007,Y 1961.237,Z 68.185,A 87.94718,B 0.00000,C 180.00000} ; retreat
  ; Step 892, bar 2119
  LIN {X 1125.007,Y 1961.237,Z 950.053,A 87.94718,B 0.00000,C 180.00000} ; outside
  LIN {X 1125.007,Y 1961.237,Z 18.185,A 87.94718,B 0.00000,C 180.00000} ; preinsert
  LIN {X 1125.007,Y 1961.237,Z -231.815,A 87.94718,B 0.00000,C 180.00000} ; insert
  LIN {X 1125.007,Y 1961.237,Z -231.815,A 87.94718,B 0.00000,C 180.00000} ; release
  LIN {X 1125.007,Y 1961.237,Z 68.185,A 87.94718,B 0.00000,C 180.00000} ; retreat
  ; Step 893, bar 2125
  LIN {X 1875.007,Y 1961.237,Z 950.053,A 87.94718,B 0.00000,C 180.00000} ; outside
  LIN {X 1875.007,Y 1961.237,Z 18.185,A 87.94718,B 0.00000,C 180.00000} ; preinsert
  LIN {X 1875.007,Y 1961.237,Z -231.815,A 87.94718,B 0.00000,C 180.00000} ; insert
  LIN {X 1875.007,Y 1961.237,Z -231.815,A 87.94718,B 0.00000,C 180.00000} ; release
  LIN {X 1875.007,Y 1961.237,Z 68.185,A 87.94718,B 0.00000,C 180.00000} ; retreat
  ; Step 894, bar 2131
  LIN {X 2625.007,Y 1961.237,Z 950.053,A 87.94718,B 0.00000,C 180.00000} ; outside
  LIN {X 2625.007,Y 1961.237,Z 18.185,A 87.94718,B 0.00000,C 180.00000} ; preinsert
  LIN {X 2625.007,Y 1961.237,Z -231.815,A 87.94718,B 0.00000,C 180.00000} ; insert
  LIN {X 2625.007,Y 1961.237,Z -231.815,A 87.94718,B 0.00000,C 180.00000} ; release
  LIN {X 2625.007,Y 1961.237,Z 68.185,A 87.94718,B 0.00000,C 180.00000} ; retreat
  ; Step 895, bar 2137
  LIN {X 3375.007,Y 1961.237,Z 950.053,A 87.94718,B 0.00000,C 180.00000} ; outside
  LIN {X 3375.007,Y 1961.237,Z 18.185,A 87.94718,B 0.00000,C 180.00000} ; preinsert
  LIN {X 3375.007,Y 1961.237,Z -231.815,A 87.94718,B 0.00000,C 180.00000} ; insert
  LIN {X 3375.007,Y 1961.237,Z -231.815,A 87.94718,B 0.00000,C 180.00000} ; release
  LIN {X 3375.007,Y 1961.237,Z 68.185,A 87.94718,B 0.00000,C 180.00000} ; retreat
  ; Step 896, bar 2143
  LIN {X 4125.007,Y 1961.237,Z 950.053,A 87.94718,B 0.00000,C 180.00000} ; outside
  LIN {X 4125.007,Y 1961.237,Z 18.185,A 87.94718,B 0.00000,C 180.00000} ; preinsert
  LIN {X 4125.007,Y 1961.237,Z -231.815,A 87.94718,B 0.00000,C 180.00000} ; insert
  LIN {X 4125.007,Y 1961.237,Z -231.815,A 87.94718,B 0.00000,C 180.00000} ; release
  LIN {X 4125.007,Y 1961.237,Z 68.185,A 87.94718,B 0.00000,C 180.00000} ; retreat
  ; Step 897, bar 2149
  LIN {X 4875.007,Y 1961.237,Z 950.053,A 87.94718,B 0.00000,C 180.00000} ; outside
  LIN {X 4875.007,Y 1961.237,Z 18.185,A 87.94718,B 0.00000,C 180.00000} ; preinsert
  LIN {X 4875.007,Y 1961.237,Z -231.815,A 87.94718,B 0.00000,C 180.00000} ; insert
  LIN {X 4875.007,Y 1961.237,Z -231.815,A 87.94718,B 0.00000,C 180.00000} ; release
  LIN {X 4875.007,Y 1961.237,Z 68.185,A 87.94718,B 0.00000,C 180.00000} ; retreat
  ; Step 898, bar 2155
  LIN {X 5625.007,Y 1961.237,Z 950.053,A 87.94718,B 0.00000,C 180.00000} ; outside
  LIN {X 5625.007,Y 1961.237,Z 18.185,A 87.94718,B 0.00000,C 180.00000} ; preinsert
  LIN {X 5625.007,Y 1961.237,Z -231.815,A 87.94718,B 0.00000,C 180.00000} ; insert
  LIN {X 5625.007,Y 1961.237,Z -231.815,A 87.94718,B 0.00000,C 180.00000} ; release
  LIN {X 5625.007,Y 1961.237,Z 68.185,A 87.94718,B 0.00000,C 180.00000} ; retreat
  ; Step 899, bar 2161
  LIN {X 6375.007,Y 1961.237,Z 950.053,A 87.94718,B 0.00000,C 180.00000} ; outside
  LIN {X 6375.007,Y 1961.237,Z 18.185,A 87.94718,B 0.00000,C 180.00000} ; preinsert
  LIN {X 6375.007,Y 1961.237,Z -231.815,A 87.94718,B 0.00000,C 180.00000} ; insert
  LIN {X 6375.007,Y 1961.237,Z -231.815,A 87.94718,B 0.00000,C 180.00000} ; release
  LIN {X 6375.007,Y 1961.237,Z 68.185,A 87.94718,B 0.00000,C 180.00000} ; retreat
  ; Step 900, bar 2167
  LIN {X 7125.007,Y 1961.237,Z 950.053,A 87.94718,B 0.00000,C 180.00000} ; outside
  LIN {X 7125.007,Y 1961.237,Z 18.185,A 87.94718,B 0.00000,C 180.00000} ; preinsert
  LIN {X 7125.007,Y 1961.237,Z -231.815,A 87.94718,B 0.00000,C 180.00000} ; insert
  LIN {X 7125.007,Y 1961.237,Z -231.815,A 87.94718,B 0.00000,C 180.00000} ; release
  LIN {X 7125.007,Y 1961.237,Z 68.185,A 87.94718,B 0.00000,C 180.00000} ; retreat
  ; Step 901, bar 2173
  LIN {X 7875.007,Y 1961.237,Z 950.053,A 87.94718,B 0.00000,C 180.00000} ; outside
  LIN {X 7875.007,Y 1961.237,Z 18.185,A 87.94718,B 0.00000,C 180.00000} ; preinsert
  LIN {X 7875.007,Y 1961.237,Z -231.815,A 87.94718,B 0.00000,C 180.00000} ; insert
  LIN {X 7875.007,Y 1961.237,Z -231.815,A 87.94718,B 0.00000,C 180.00000} ; release
  LIN {X 7875.007,Y 1961.237,Z 68.185,A 87.94718,B 0.00000,C 180.00000} ; retreat
  ; Step 902, bar 2179
  LIN {X 8625.007,Y 1961.237,Z 950.053,A 87.94718,B 0.00000,C 180.00000} ; outside
  LIN {X 8625.007,Y 1961.237,Z 18.185,A 87.94718,B 0.00000,C 180.00000} ; preinsert
  LIN {X 8625.007,Y 1961.237,Z -231.815,A 87.94718,B 0.00000,C 180.00000} ; insert
  LIN {X 8625.007,Y 1961.237,Z -231.815,A 87.94718,B 0.00000,C 180.00000} ; release
  LIN {X 8625.007,Y 1961.237,Z 68.185,A 87.94718,B 0.00000,C 180.00000} ; retreat
  ; Step 903, bar 2185
  LIN {X 9375.007,Y 1961.237,Z 950.053,A 87.94718,B 0.00000,C 180.00000} ; outside
  LIN {X 9375.007,Y 1961.237,Z 18.185,A 87.94718,B 0.00000,C 180.00000} ; preinsert
  LIN {X 9375.007,Y 1961.237,Z -231.815,A 87.94718,B 0.00000,C 180.00000} ; insert
  LIN {X 9375.007,Y 1961.237,Z -231.815,A 87.94718,B 0.00000,C 180.00000} ; release
  LIN {X 9375.007,Y 1961.237,Z 68.185,A 87.94718,B 0.00000,C 180.00000} ; retreat
  ; Step 904, bar 2191
  LIN {X 10125.007,Y 1961.237,Z 950.053,A 87.94718,B 0.00000,C 180.00000} ; outside
  LIN {X 10125.007,Y 1961.237,Z 18.185,A 87.94718,B 0.00000,C 180.00000} ; preinsert
  LIN {X 10125.007,Y 1961.237,Z -231.815,A 87.94718,B 0.00000,C 180.00000} ; insert
  LIN {X 10125.007,Y 1961.237,Z -231.815,A 87.94718,B 0.00000,C 180.00000} ; release
  LIN {X 10125.007,Y 1961.237,Z 68.185,A 87.94718,B 0.00000,C 180.00000} ; retreat
  ; Step 905, bar 2197
  LIN {X 10875.007,Y 1961.237,Z 950.053,A 87.94718,B 0.00000,C 180.00000} ; outside
  LIN {X 10875.007,Y 1961.237,Z 18.185,A 87.94718,B 0.00000,C 180.00000} ; preinsert
  LIN {X 10875.007,Y 1961.237,Z -231.815,A 87.94718,B 0.00000,C 180.00000} ; insert
  LIN {X 10875.007,Y 1961.237,Z -231.815,A 87.94718,B 0.00000,C 180.00000} ; release
  LIN {X 10875.007,Y 1961.237,Z 68.185,A 87.94718,B 0.00000,C 180.00000} ; retreat
  ; Step 906, bar 2203
  LIN {X 11625.007,Y 1961.237,Z 950.053,A 87.94718,B 0.00000,C 180.00000} ; outside
  LIN {X 11625.007,Y 1961.237,Z 18.185,A 87.94718,B 0.00000,C 180.00000} ; preinsert
  LIN {X 11625.007,Y 1961.237,Z -231.815,A 87.94718,B 0.00000,C 180.00000} ; insert
  LIN {X 11625.007,Y 1961.237,Z -231.815,A 87.94718,B 0.00000,C 180.00000} ; release
  LIN {X 11625.007,Y 1961.237,Z 68.185,A 87.94718,B 0.00000,C 180.00000} ; retreat
  ; Step 907, bar 2209
  LIN {X 12250.007,Y 1961.237,Z 950.053,A 87.94718,B 0.00000,C 180.00000} ; outside
